REGION Network 10
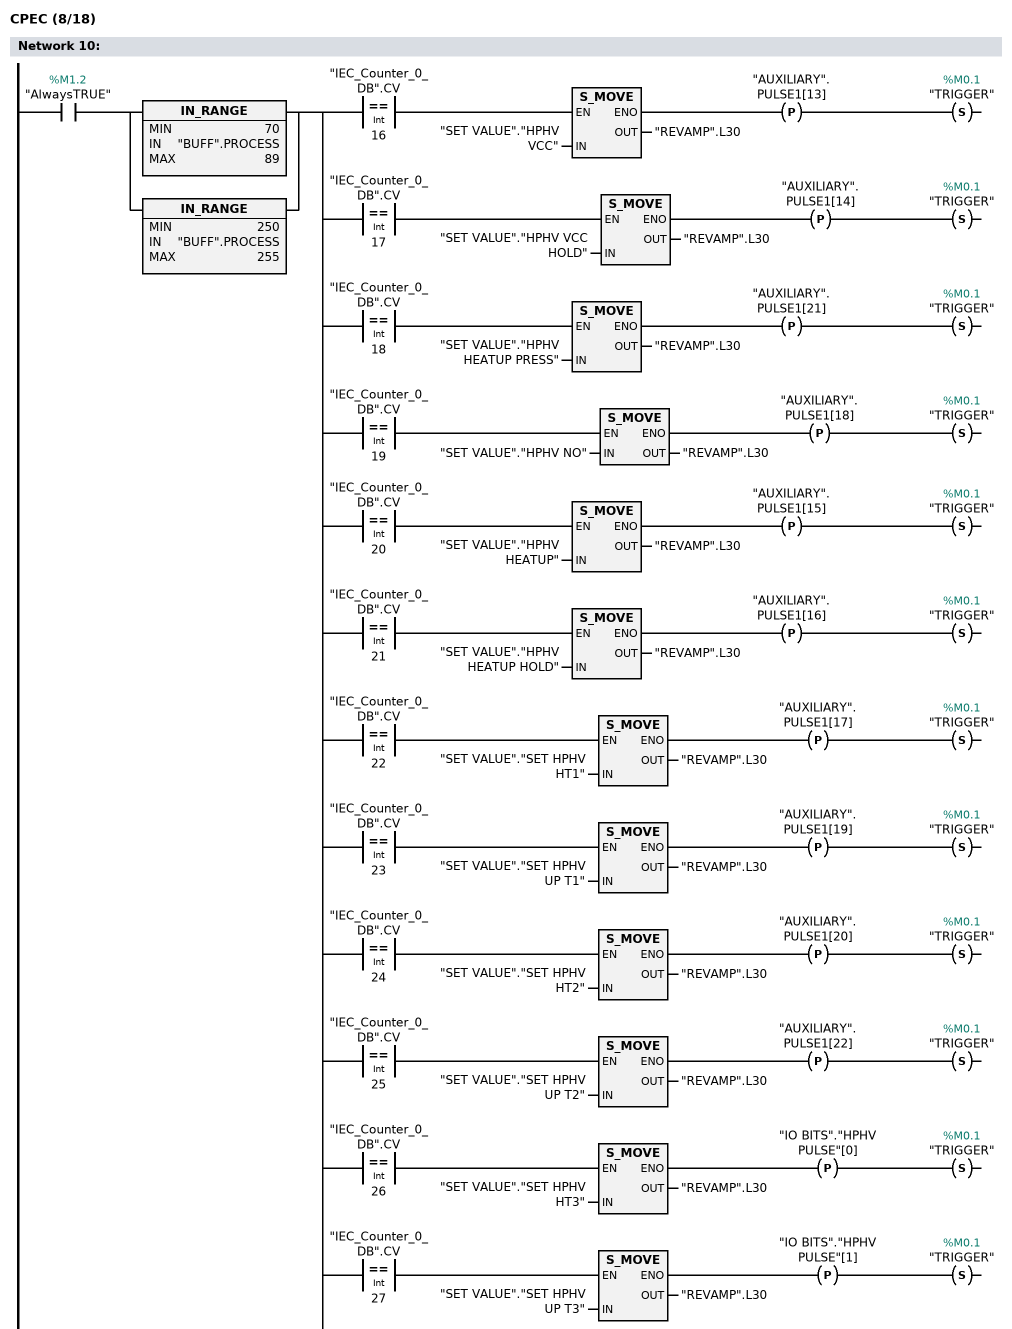
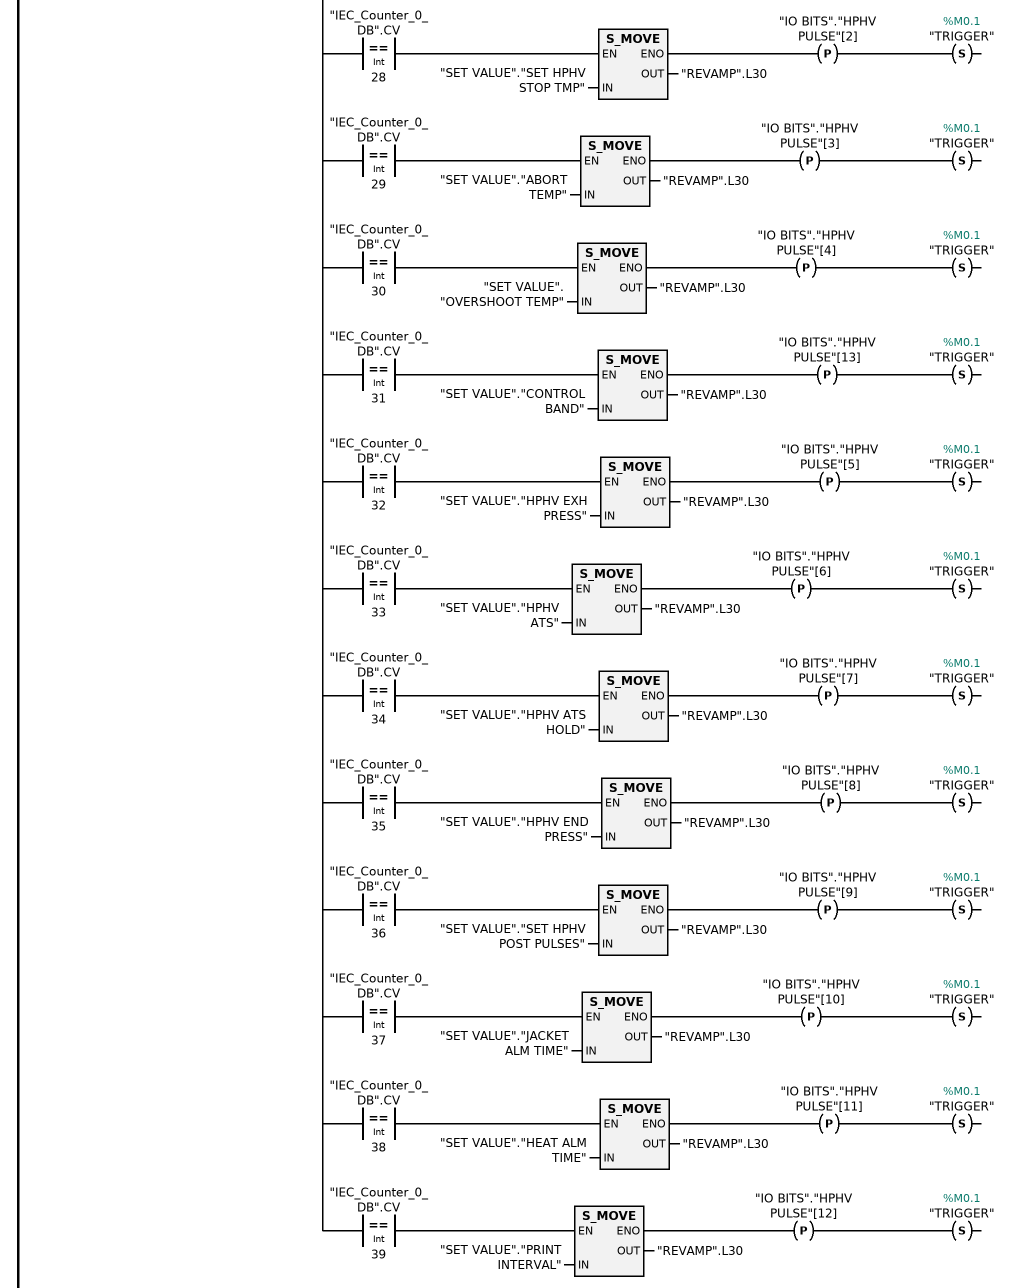
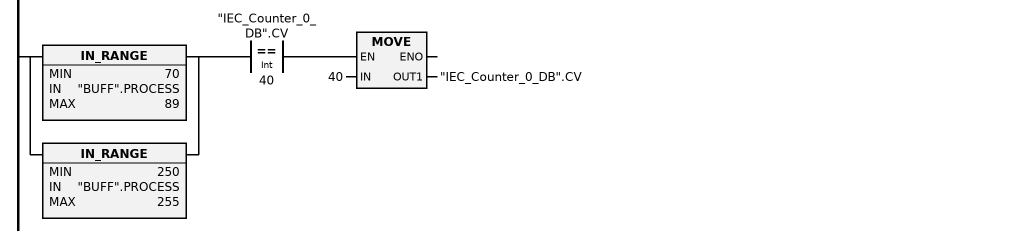
   RUNG wire#powerrail
      Contact( "AlwaysTRUE" )
      wire#w1
      { S7_Templates := "SrcType := Int" } InRange(min := 70, in := "BUFF".PROCESS, max := 89)
      wire#w2
      { S7_Templates := "SrcType := Int" } EQ_Contact(in1 := "IEC_Counter_0_DB".CV, in2 := 16)
      S_Move(in := "SET VALUE"."HPHV VCC", out => "REVAMP".L30)
      P_Trig( "AUXILIARY".PULSE1[13] )
      S_Coil( "TRIGGER" )
   END_RUNG
   RUNG wire#w1
      { S7_Templates := "SrcType := Int" } InRange(min := 250, in := "BUFF".PROCESS, max := 255)
   END_RUNG wire#w2
   RUNG wire#w2
      { S7_Templates := "SrcType := Int" } EQ_Contact(in1 := "IEC_Counter_0_DB".CV, in2 := 17)
      S_Move(in := "SET VALUE"."HPHV VCC HOLD", out => "REVAMP".L30)
      P_Trig( "AUXILIARY".PULSE1[14] )
      S_Coil( "TRIGGER" )
   END_RUNG
   RUNG wire#w2
      { S7_Templates := "SrcType := Int" } EQ_Contact(in1 := "IEC_Counter_0_DB".CV, in2 := 18)
      S_Move(in := "SET VALUE"."HPHV HEATUP PRESS", out => "REVAMP".L30)
      P_Trig( "AUXILIARY".PULSE1[21] )
      S_Coil( "TRIGGER" )
   END_RUNG
   RUNG wire#w2
      { S7_Templates := "SrcType := Int" } EQ_Contact(in1 := "IEC_Counter_0_DB".CV, in2 := 19)
      S_Move(in := "SET VALUE"."HPHV NO", out => "REVAMP".L30)
      P_Trig( "AUXILIARY".PULSE1[18] )
      S_Coil( "TRIGGER" )
   END_RUNG
   RUNG wire#w2
      { S7_Templates := "SrcType := Int" } EQ_Contact(in1 := "IEC_Counter_0_DB".CV, in2 := 20)
      S_Move(in := "SET VALUE"."HPHV HEATUP", out => "REVAMP".L30)
      P_Trig( "AUXILIARY".PULSE1[15] )
      S_Coil( "TRIGGER" )
   END_RUNG
   RUNG wire#w2
      { S7_Templates := "SrcType := Int" } EQ_Contact(in1 := "IEC_Counter_0_DB".CV, in2 := 21)
      S_Move(in := "SET VALUE"."HPHV HEATUP HOLD", out => "REVAMP".L30)
      P_Trig( "AUXILIARY".PULSE1[16] )
      S_Coil( "TRIGGER" )
   END_RUNG
   RUNG wire#w2
      { S7_Templates := "SrcType := Int" } EQ_Contact(in1 := "IEC_Counter_0_DB".CV, in2 := 22)
      S_Move(in := "SET VALUE"."SET HPHV HT1", out => "REVAMP".L30)
      P_Trig( "AUXILIARY".PULSE1[17] )
      S_Coil( "TRIGGER" )
   END_RUNG
   RUNG wire#w2
      { S7_Templates := "SrcType := Int" } EQ_Contact(in1 := "IEC_Counter_0_DB".CV, in2 := 23)
      S_Move(in := "SET VALUE"."SET HPHV UP T1", out => "REVAMP".L30)
      P_Trig( "AUXILIARY".PULSE1[19] )
      S_Coil( "TRIGGER" )
   END_RUNG
   RUNG wire#w2
      { S7_Templates := "SrcType := Int" } EQ_Contact(in1 := "IEC_Counter_0_DB".CV, in2 := 24)
      S_Move(in := "SET VALUE"."SET HPHV HT2", out => "REVAMP".L30)
      P_Trig( "AUXILIARY".PULSE1[20] )
      S_Coil( "TRIGGER" )
   END_RUNG
   RUNG wire#w2
      { S7_Templates := "SrcType := Int" } EQ_Contact(in1 := "IEC_Counter_0_DB".CV, in2 := 25)
      S_Move(in := "SET VALUE"."SET HPHV UP T2", out => "REVAMP".L30)
      P_Trig( "AUXILIARY".PULSE1[22] )
      S_Coil( "TRIGGER" )
   END_RUNG
   RUNG wire#w2
      { S7_Templates := "SrcType := Int" } EQ_Contact(in1 := "IEC_Counter_0_DB".CV, in2 := 26)
      S_Move(in := "SET VALUE"."SET HPHV HT3", out => "REVAMP".L30)
      P_Trig( "IO BITS"."HPHV PULSE"[0] )
      S_Coil( "TRIGGER" )
   END_RUNG
   RUNG wire#w2
      { S7_Templates := "SrcType := Int" } EQ_Contact(in1 := "IEC_Counter_0_DB".CV, in2 := 27)
      S_Move(in := "SET VALUE"."SET HPHV UP T3", out => "REVAMP".L30)
      P_Trig( "IO BITS"."HPHV PULSE"[1] )
      S_Coil( "TRIGGER" )
   END_RUNG
   RUNG wire#w2
      { S7_Templates := "SrcType := Int" } EQ_Contact(in1 := "IEC_Counter_0_DB".CV, in2 := 28)
      S_Move(in := "SET VALUE"."SET HPHV STOP TMP", out => "REVAMP".L30)
      P_Trig( "IO BITS"."HPHV PULSE"[2] )
      S_Coil( "TRIGGER" )
   END_RUNG
   RUNG wire#w2
      { S7_Templates := "SrcType := Int" } EQ_Contact(in1 := "IEC_Counter_0_DB".CV, in2 := 29)
      S_Move(in := "SET VALUE"."ABORT TEMP", out => "REVAMP".L30)
      P_Trig( "IO BITS"."HPHV PULSE"[3] )
      S_Coil( "TRIGGER" )
   END_RUNG
   RUNG wire#w2
      { S7_Templates := "SrcType := Int" } EQ_Contact(in1 := "IEC_Counter_0_DB".CV, in2 := 30)
      S_Move(in := "SET VALUE"."OVERSHOOT TEMP", out => "REVAMP".L30)
      P_Trig( "IO BITS"."HPHV PULSE"[4] )
      S_Coil( "TRIGGER" )
   END_RUNG
   RUNG wire#w2
      { S7_Templates := "SrcType := Int" } EQ_Contact(in1 := "IEC_Counter_0_DB".CV, in2 := 31)
      S_Move(in := "SET VALUE"."CONTROL BAND", out => "REVAMP".L30)
      P_Trig( "IO BITS"."HPHV PULSE"[13] )
      S_Coil( "TRIGGER" )
   END_RUNG
   RUNG wire#w2
      { S7_Templates := "SrcType := Int" } EQ_Contact(in1 := "IEC_Counter_0_DB".CV, in2 := 32)
      S_Move(in := "SET VALUE"."HPHV EXH PRESS", out => "REVAMP".L30)
      P_Trig( "IO BITS"."HPHV PULSE"[5] )
      S_Coil( "TRIGGER" )
   END_RUNG
   RUNG wire#w2
      { S7_Templates := "SrcType := Int" } EQ_Contact(in1 := "IEC_Counter_0_DB".CV, in2 := 33)
      S_Move(in := "SET VALUE"."HPHV ATS", out => "REVAMP".L30)
      P_Trig( "IO BITS"."HPHV PULSE"[6] )
      S_Coil( "TRIGGER" )
   END_RUNG
   RUNG wire#w2
      { S7_Templates := "SrcType := Int" } EQ_Contact(in1 := "IEC_Counter_0_DB".CV, in2 := 34)
      S_Move(in := "SET VALUE"."HPHV ATS HOLD", out => "REVAMP".L30)
      P_Trig( "IO BITS"."HPHV PULSE"[7] )
      S_Coil( "TRIGGER" )
   END_RUNG
   RUNG wire#w2
      { S7_Templates := "SrcType := Int" } EQ_Contact(in1 := "IEC_Counter_0_DB".CV, in2 := 35)
      S_Move(in := "SET VALUE"."HPHV END PRESS", out => "REVAMP".L30)
      P_Trig( "IO BITS"."HPHV PULSE"[8] )
      S_Coil( "TRIGGER" )
   END_RUNG
   RUNG wire#w2
      { S7_Templates := "SrcType := Int" } EQ_Contact(in1 := "IEC_Counter_0_DB".CV, in2 := 36)
      S_Move(in := "SET VALUE"."SET HPHV POST PULSES", out => "REVAMP".L30)
      P_Trig( "IO BITS"."HPHV PULSE"[9] )
      S_Coil( "TRIGGER" )
   END_RUNG
   RUNG wire#w2
      { S7_Templates := "SrcType := Int" } EQ_Contact(in1 := "IEC_Counter_0_DB".CV, in2 := 37)
      S_Move(in := "SET VALUE"."JACKET ALM TIME", out => "REVAMP".L30)
      P_Trig( "IO BITS"."HPHV PULSE"[10] )
      S_Coil( "TRIGGER" )
   END_RUNG
   RUNG wire#w2
      { S7_Templates := "SrcType := Int" } EQ_Contact(in1 := "IEC_Counter_0_DB".CV, in2 := 38)
      S_Move(in := "SET VALUE"."HEAT ALM TIME", out => "REVAMP".L30)
      P_Trig( "IO BITS"."HPHV PULSE"[11] )
      S_Coil( "TRIGGER" )
   END_RUNG
   RUNG wire#w2
      { S7_Templates := "SrcType := Int" } EQ_Contact(in1 := "IEC_Counter_0_DB".CV, in2 := 39)
      S_Move(in := "SET VALUE"."PRINT INTERVAL", out => "REVAMP".L30)
      P_Trig( "IO BITS"."HPHV PULSE"[12] )
      S_Coil( "TRIGGER" )
   END_RUNG
   RUNG wire#powerrail
      { S7_Templates := "SrcType := Int" } InRange(min := 70, in := "BUFF".PROCESS, max := 89)
      wire#w3
      { S7_Templates := "SrcType := Int" } EQ_Contact(in1 := "IEC_Counter_0_DB".CV, in2 := 40)
      Move(in := 40, out1 => "IEC_Counter_0_DB".CV)
   END_RUNG
   RUNG wire#powerrail
      { S7_Templates := "SrcType := Int" } InRange(min := 250, in := "BUFF".PROCESS, max := 255)
   END_RUNG wire#w3
   // the same network as SCL:
   #_w1 := "AlwaysTRUE" AND (((70 <= "BUFF".PROCESS) AND ("BUFF".PROCESS <= 89)) OR ((250 <= "BUFF".PROCESS) AND ("BUFF".PROCESS <= 255)));
   #_w2 := #_w1 AND ("IEC_Counter_0_DB".CV = 16);
   IF #_w2 THEN "REVAMP".L30 := "SET VALUE"."HPHV VCC"; END_IF;
   #_w3 := #_w2 AND NOT "AUXILIARY".PULSE1[13];   // rising edge
   "AUXILIARY".PULSE1[13] := #_w2;
   IF #_w3 THEN "TRIGGER" := TRUE; END_IF;
   #_w4 := #_w1 AND ("IEC_Counter_0_DB".CV = 17);
   IF #_w4 THEN "REVAMP".L30 := "SET VALUE"."HPHV VCC HOLD"; END_IF;
   #_w5 := #_w4 AND NOT "AUXILIARY".PULSE1[14];   // rising edge
   "AUXILIARY".PULSE1[14] := #_w4;
   IF #_w5 THEN "TRIGGER" := TRUE; END_IF;
   #_w6 := #_w1 AND ("IEC_Counter_0_DB".CV = 18);
   IF #_w6 THEN "REVAMP".L30 := "SET VALUE"."HPHV HEATUP PRESS"; END_IF;
   #_w7 := #_w6 AND NOT "AUXILIARY".PULSE1[21];   // rising edge
   "AUXILIARY".PULSE1[21] := #_w6;
   IF #_w7 THEN "TRIGGER" := TRUE; END_IF;
   #_w8 := #_w1 AND ("IEC_Counter_0_DB".CV = 19);
   IF #_w8 THEN "REVAMP".L30 := "SET VALUE"."HPHV NO"; END_IF;
   #_w9 := #_w8 AND NOT "AUXILIARY".PULSE1[18];   // rising edge
   "AUXILIARY".PULSE1[18] := #_w8;
   IF #_w9 THEN "TRIGGER" := TRUE; END_IF;
   #_w10 := #_w1 AND ("IEC_Counter_0_DB".CV = 20);
   IF #_w10 THEN "REVAMP".L30 := "SET VALUE"."HPHV HEATUP"; END_IF;
   #_w11 := #_w10 AND NOT "AUXILIARY".PULSE1[15];   // rising edge
   "AUXILIARY".PULSE1[15] := #_w10;
   IF #_w11 THEN "TRIGGER" := TRUE; END_IF;
   #_w12 := #_w1 AND ("IEC_Counter_0_DB".CV = 21);
   IF #_w12 THEN "REVAMP".L30 := "SET VALUE"."HPHV HEATUP HOLD"; END_IF;
   #_w13 := #_w12 AND NOT "AUXILIARY".PULSE1[16];   // rising edge
   "AUXILIARY".PULSE1[16] := #_w12;
   IF #_w13 THEN "TRIGGER" := TRUE; END_IF;
   #_w14 := #_w1 AND ("IEC_Counter_0_DB".CV = 22);
   IF #_w14 THEN "REVAMP".L30 := "SET VALUE"."SET HPHV HT1"; END_IF;
   #_w15 := #_w14 AND NOT "AUXILIARY".PULSE1[17];   // rising edge
   "AUXILIARY".PULSE1[17] := #_w14;
   IF #_w15 THEN "TRIGGER" := TRUE; END_IF;
   #_w16 := #_w1 AND ("IEC_Counter_0_DB".CV = 23);
   IF #_w16 THEN "REVAMP".L30 := "SET VALUE"."SET HPHV UP T1"; END_IF;
   #_w17 := #_w16 AND NOT "AUXILIARY".PULSE1[19];   // rising edge
   "AUXILIARY".PULSE1[19] := #_w16;
   IF #_w17 THEN "TRIGGER" := TRUE; END_IF;
   #_w18 := #_w1 AND ("IEC_Counter_0_DB".CV = 24);
   IF #_w18 THEN "REVAMP".L30 := "SET VALUE"."SET HPHV HT2"; END_IF;
   #_w19 := #_w18 AND NOT "AUXILIARY".PULSE1[20];   // rising edge
   "AUXILIARY".PULSE1[20] := #_w18;
   IF #_w19 THEN "TRIGGER" := TRUE; END_IF;
   #_w20 := #_w1 AND ("IEC_Counter_0_DB".CV = 25);
   IF #_w20 THEN "REVAMP".L30 := "SET VALUE"."SET HPHV UP T2"; END_IF;
   #_w21 := #_w20 AND NOT "AUXILIARY".PULSE1[22];   // rising edge
   "AUXILIARY".PULSE1[22] := #_w20;
   IF #_w21 THEN "TRIGGER" := TRUE; END_IF;
   #_w22 := #_w1 AND ("IEC_Counter_0_DB".CV = 26);
   IF #_w22 THEN "REVAMP".L30 := "SET VALUE"."SET HPHV HT3"; END_IF;
   #_w23 := #_w22 AND NOT "IO BITS"."HPHV PULSE"[0];   // rising edge
   "IO BITS"."HPHV PULSE"[0] := #_w22;
   IF #_w23 THEN "TRIGGER" := TRUE; END_IF;
   #_w24 := #_w1 AND ("IEC_Counter_0_DB".CV = 27);
   IF #_w24 THEN "REVAMP".L30 := "SET VALUE"."SET HPHV UP T3"; END_IF;
   #_w25 := #_w24 AND NOT "IO BITS"."HPHV PULSE"[1];   // rising edge
   "IO BITS"."HPHV PULSE"[1] := #_w24;
   IF #_w25 THEN "TRIGGER" := TRUE; END_IF;
   #_w26 := #_w1 AND ("IEC_Counter_0_DB".CV = 28);
   IF #_w26 THEN "REVAMP".L30 := "SET VALUE"."SET HPHV STOP TMP"; END_IF;
   #_w27 := #_w26 AND NOT "IO BITS"."HPHV PULSE"[2];   // rising edge
   "IO BITS"."HPHV PULSE"[2] := #_w26;
   IF #_w27 THEN "TRIGGER" := TRUE; END_IF;
   #_w28 := #_w1 AND ("IEC_Counter_0_DB".CV = 29);
   IF #_w28 THEN "REVAMP".L30 := "SET VALUE"."ABORT TEMP"; END_IF;
   #_w29 := #_w28 AND NOT "IO BITS"."HPHV PULSE"[3];   // rising edge
   "IO BITS"."HPHV PULSE"[3] := #_w28;
   IF #_w29 THEN "TRIGGER" := TRUE; END_IF;
   #_w30 := #_w1 AND ("IEC_Counter_0_DB".CV = 30);
   IF #_w30 THEN "REVAMP".L30 := "SET VALUE"."OVERSHOOT TEMP"; END_IF;
   #_w31 := #_w30 AND NOT "IO BITS"."HPHV PULSE"[4];   // rising edge
   "IO BITS"."HPHV PULSE"[4] := #_w30;
   IF #_w31 THEN "TRIGGER" := TRUE; END_IF;
   #_w32 := #_w1 AND ("IEC_Counter_0_DB".CV = 31);
   IF #_w32 THEN "REVAMP".L30 := "SET VALUE"."CONTROL BAND"; END_IF;
   #_w33 := #_w32 AND NOT "IO BITS"."HPHV PULSE"[13];   // rising edge
   "IO BITS"."HPHV PULSE"[13] := #_w32;
   IF #_w33 THEN "TRIGGER" := TRUE; END_IF;
   #_w34 := #_w1 AND ("IEC_Counter_0_DB".CV = 32);
   IF #_w34 THEN "REVAMP".L30 := "SET VALUE"."HPHV EXH PRESS"; END_IF;
   #_w35 := #_w34 AND NOT "IO BITS"."HPHV PULSE"[5];   // rising edge
   "IO BITS"."HPHV PULSE"[5] := #_w34;
   IF #_w35 THEN "TRIGGER" := TRUE; END_IF;
   #_w36 := #_w1 AND ("IEC_Counter_0_DB".CV = 33);
   IF #_w36 THEN "REVAMP".L30 := "SET VALUE"."HPHV ATS"; END_IF;
   #_w37 := #_w36 AND NOT "IO BITS"."HPHV PULSE"[6];   // rising edge
   "IO BITS"."HPHV PULSE"[6] := #_w36;
   IF #_w37 THEN "TRIGGER" := TRUE; END_IF;
   #_w38 := #_w1 AND ("IEC_Counter_0_DB".CV = 34);
   IF #_w38 THEN "REVAMP".L30 := "SET VALUE"."HPHV ATS HOLD"; END_IF;
   #_w39 := #_w38 AND NOT "IO BITS"."HPHV PULSE"[7];   // rising edge
   "IO BITS"."HPHV PULSE"[7] := #_w38;
   IF #_w39 THEN "TRIGGER" := TRUE; END_IF;
   #_w40 := #_w1 AND ("IEC_Counter_0_DB".CV = 35);
   IF #_w40 THEN "REVAMP".L30 := "SET VALUE"."HPHV END PRESS"; END_IF;
   #_w41 := #_w40 AND NOT "IO BITS"."HPHV PULSE"[8];   // rising edge
   "IO BITS"."HPHV PULSE"[8] := #_w40;
   IF #_w41 THEN "TRIGGER" := TRUE; END_IF;
   #_w42 := #_w1 AND ("IEC_Counter_0_DB".CV = 36);
   IF #_w42 THEN "REVAMP".L30 := "SET VALUE"."SET HPHV POST PULSES"; END_IF;
   #_w43 := #_w42 AND NOT "IO BITS"."HPHV PULSE"[9];   // rising edge
   "IO BITS"."HPHV PULSE"[9] := #_w42;
   IF #_w43 THEN "TRIGGER" := TRUE; END_IF;
   #_w44 := #_w1 AND ("IEC_Counter_0_DB".CV = 37);
   IF #_w44 THEN "REVAMP".L30 := "SET VALUE"."JACKET ALM TIME"; END_IF;
   #_w45 := #_w44 AND NOT "IO BITS"."HPHV PULSE"[10];   // rising edge
   "IO BITS"."HPHV PULSE"[10] := #_w44;
   IF #_w45 THEN "TRIGGER" := TRUE; END_IF;
   #_w46 := #_w1 AND ("IEC_Counter_0_DB".CV = 38);
   IF #_w46 THEN "REVAMP".L30 := "SET VALUE"."HEAT ALM TIME"; END_IF;
   #_w47 := #_w46 AND NOT "IO BITS"."HPHV PULSE"[11];   // rising edge
   "IO BITS"."HPHV PULSE"[11] := #_w46;
   IF #_w47 THEN "TRIGGER" := TRUE; END_IF;
   #_w48 := #_w1 AND ("IEC_Counter_0_DB".CV = 39);
   IF #_w48 THEN "REVAMP".L30 := "SET VALUE"."PRINT INTERVAL"; END_IF;
   #_w49 := #_w48 AND NOT "IO BITS"."HPHV PULSE"[12];   // rising edge
   "IO BITS"."HPHV PULSE"[12] := #_w48;
   IF #_w49 THEN "TRIGGER" := TRUE; END_IF;
   IF (((70 <= "BUFF".PROCESS) AND ("BUFF".PROCESS <= 89)) OR ((250 <= "BUFF".PROCESS) AND ("BUFF".PROCESS <= 255))) AND ("IEC_Counter_0_DB".CV = 40) THEN
       "IEC_Counter_0_DB".CV := 40;
   END_IF;
END_REGION

REGION Network 11
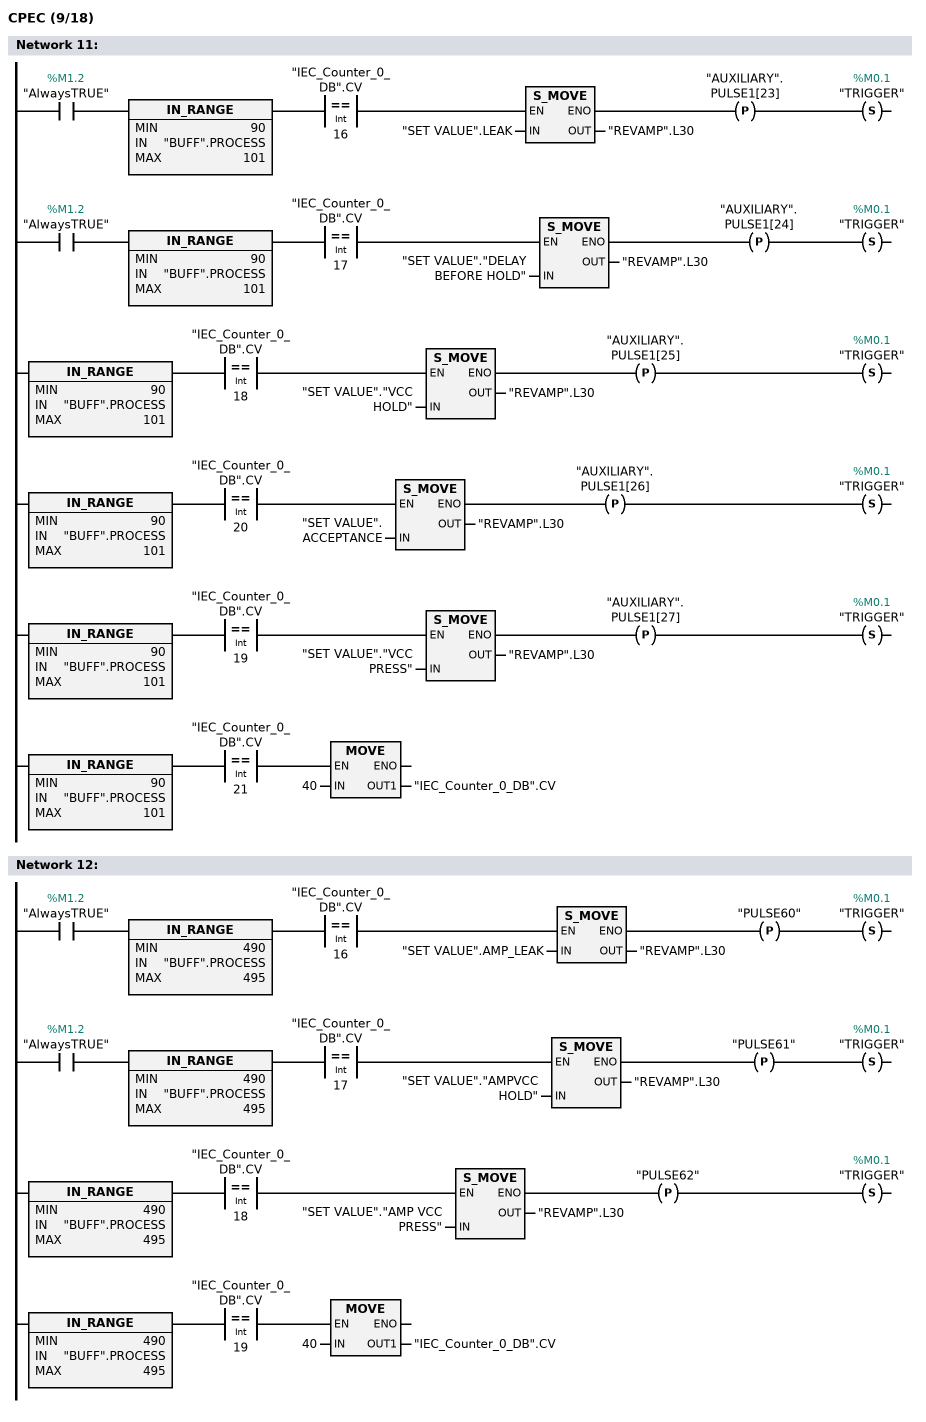
   RUNG wire#powerrail
      Contact( "AlwaysTRUE" )
      { S7_Templates := "SrcType := Int" } InRange(min := 90, in := "BUFF".PROCESS, max := 101)
      { S7_Templates := "SrcType := Int" } EQ_Contact(in1 := "IEC_Counter_0_DB".CV, in2 := 16)
      S_Move(in := "SET VALUE".LEAK, out => "REVAMP".L30)
      P_Trig( "AUXILIARY".PULSE1[23] )
      S_Coil( "TRIGGER" )
   END_RUNG
   RUNG wire#powerrail
      Contact( "AlwaysTRUE" )
      { S7_Templates := "SrcType := Int" } InRange(min := 90, in := "BUFF".PROCESS, max := 101)
      { S7_Templates := "SrcType := Int" } EQ_Contact(in1 := "IEC_Counter_0_DB".CV, in2 := 17)
      S_Move(in := "SET VALUE"."DELAY BEFORE HOLD", out => "REVAMP".L30)
      P_Trig( "AUXILIARY".PULSE1[24] )
      S_Coil( "TRIGGER" )
   END_RUNG
   RUNG wire#powerrail
      { S7_Templates := "SrcType := Int" } InRange(min := 90, in := "BUFF".PROCESS, max := 101)
      { S7_Templates := "SrcType := Int" } EQ_Contact(in1 := "IEC_Counter_0_DB".CV, in2 := 18)
      S_Move(in := "SET VALUE"."VCC HOLD", out => "REVAMP".L30)
      P_Trig( "AUXILIARY".PULSE1[25] )
      S_Coil( "TRIGGER" )
   END_RUNG
   RUNG wire#powerrail
      { S7_Templates := "SrcType := Int" } InRange(min := 90, in := "BUFF".PROCESS, max := 101)
      { S7_Templates := "SrcType := Int" } EQ_Contact(in1 := "IEC_Counter_0_DB".CV, in2 := 20)
      S_Move(in := "SET VALUE".ACCEPTANCE, out => "REVAMP".L30)
      P_Trig( "AUXILIARY".PULSE1[26] )
      S_Coil( "TRIGGER" )
   END_RUNG
   RUNG wire#powerrail
      { S7_Templates := "SrcType := Int" } InRange(min := 90, in := "BUFF".PROCESS, max := 101)
      { S7_Templates := "SrcType := Int" } EQ_Contact(in1 := "IEC_Counter_0_DB".CV, in2 := 19)
      S_Move(in := "SET VALUE"."VCC PRESS", out => "REVAMP".L30)
      P_Trig( "AUXILIARY".PULSE1[27] )
      S_Coil( "TRIGGER" )
   END_RUNG
   RUNG wire#powerrail
      { S7_Templates := "SrcType := Int" } InRange(min := 90, in := "BUFF".PROCESS, max := 101)
      { S7_Templates := "SrcType := Int" } EQ_Contact(in1 := "IEC_Counter_0_DB".CV, in2 := 21)
      Move(in := 40, out1 => "IEC_Counter_0_DB".CV)
   END_RUNG
   // the same network as SCL:
   #_w1 := "AlwaysTRUE" AND (90 <= "BUFF".PROCESS) AND ("BUFF".PROCESS <= 101) AND ("IEC_Counter_0_DB".CV = 16);
   IF #_w1 THEN "REVAMP".L30 := "SET VALUE".LEAK; END_IF;
   #_w2 := #_w1 AND NOT "AUXILIARY".PULSE1[23];   // rising edge
   "AUXILIARY".PULSE1[23] := #_w1;
   IF #_w2 THEN "TRIGGER" := TRUE; END_IF;
   #_w3 := "AlwaysTRUE" AND (90 <= "BUFF".PROCESS) AND ("BUFF".PROCESS <= 101) AND ("IEC_Counter_0_DB".CV = 17);
   IF #_w3 THEN "REVAMP".L30 := "SET VALUE"."DELAY BEFORE HOLD"; END_IF;
   #_w4 := #_w3 AND NOT "AUXILIARY".PULSE1[24];   // rising edge
   "AUXILIARY".PULSE1[24] := #_w3;
   IF #_w4 THEN "TRIGGER" := TRUE; END_IF;
   #_w5 := (90 <= "BUFF".PROCESS) AND ("BUFF".PROCESS <= 101) AND ("IEC_Counter_0_DB".CV = 18);
   IF #_w5 THEN "REVAMP".L30 := "SET VALUE"."VCC HOLD"; END_IF;
   #_w6 := #_w5 AND NOT "AUXILIARY".PULSE1[25];   // rising edge
   "AUXILIARY".PULSE1[25] := #_w5;
   IF #_w6 THEN "TRIGGER" := TRUE; END_IF;
   #_w7 := (90 <= "BUFF".PROCESS) AND ("BUFF".PROCESS <= 101) AND ("IEC_Counter_0_DB".CV = 20);
   IF #_w7 THEN "REVAMP".L30 := "SET VALUE".ACCEPTANCE; END_IF;
   #_w8 := #_w7 AND NOT "AUXILIARY".PULSE1[26];   // rising edge
   "AUXILIARY".PULSE1[26] := #_w7;
   IF #_w8 THEN "TRIGGER" := TRUE; END_IF;
   #_w9 := (90 <= "BUFF".PROCESS) AND ("BUFF".PROCESS <= 101) AND ("IEC_Counter_0_DB".CV = 19);
   IF #_w9 THEN "REVAMP".L30 := "SET VALUE"."VCC PRESS"; END_IF;
   #_w10 := #_w9 AND NOT "AUXILIARY".PULSE1[27];   // rising edge
   "AUXILIARY".PULSE1[27] := #_w9;
   IF #_w10 THEN "TRIGGER" := TRUE; END_IF;
   IF (90 <= "BUFF".PROCESS) AND ("BUFF".PROCESS <= 101) AND ("IEC_Counter_0_DB".CV = 21) THEN
       "IEC_Counter_0_DB".CV := 40;
   END_IF;
END_REGION

REGION Network 12
   RUNG wire#powerrail
      Contact( "AlwaysTRUE" )
      { S7_Templates := "SrcType := Int" } InRange(min := 490, in := "BUFF".PROCESS, max := 495)
      { S7_Templates := "SrcType := Int" } EQ_Contact(in1 := "IEC_Counter_0_DB".CV, in2 := 16)
      S_Move(in := "SET VALUE".AMP_LEAK, out => "REVAMP".L30)
      P_Trig( "PULSE60" )
      S_Coil( "TRIGGER" )
   END_RUNG
   RUNG wire#powerrail
      Contact( "AlwaysTRUE" )
      { S7_Templates := "SrcType := Int" } InRange(min := 490, in := "BUFF".PROCESS, max := 495)
      { S7_Templates := "SrcType := Int" } EQ_Contact(in1 := "IEC_Counter_0_DB".CV, in2 := 17)
      S_Move(in := "SET VALUE"."AMPVCC HOLD", out => "REVAMP".L30)
      P_Trig( "PULSE61" )
      S_Coil( "TRIGGER" )
   END_RUNG
   RUNG wire#powerrail
      { S7_Templates := "SrcType := Int" } InRange(min := 490, in := "BUFF".PROCESS, max := 495)
      { S7_Templates := "SrcType := Int" } EQ_Contact(in1 := "IEC_Counter_0_DB".CV, in2 := 18)
      S_Move(in := "SET VALUE"."AMP VCC PRESS", out => "REVAMP".L30)
      P_Trig( "PULSE62" )
      S_Coil( "TRIGGER" )
   END_RUNG
   RUNG wire#powerrail
      { S7_Templates := "SrcType := Int" } InRange(min := 490, in := "BUFF".PROCESS, max := 495)
      { S7_Templates := "SrcType := Int" } EQ_Contact(in1 := "IEC_Counter_0_DB".CV, in2 := 19)
      Move(in := 40, out1 => "IEC_Counter_0_DB".CV)
   END_RUNG
   // the same network as SCL:
   #_w1 := "AlwaysTRUE" AND (490 <= "BUFF".PROCESS) AND ("BUFF".PROCESS <= 495) AND ("IEC_Counter_0_DB".CV = 16);
   IF #_w1 THEN "REVAMP".L30 := "SET VALUE".AMP_LEAK; END_IF;
   #_w2 := #_w1 AND NOT "PULSE60";   // rising edge
   "PULSE60" := #_w1;
   IF #_w2 THEN "TRIGGER" := TRUE; END_IF;
   #_w3 := "AlwaysTRUE" AND (490 <= "BUFF".PROCESS) AND ("BUFF".PROCESS <= 495) AND ("IEC_Counter_0_DB".CV = 17);
   IF #_w3 THEN "REVAMP".L30 := "SET VALUE"."AMPVCC HOLD"; END_IF;
   #_w4 := #_w3 AND NOT "PULSE61";   // rising edge
   "PULSE61" := #_w3;
   IF #_w4 THEN "TRIGGER" := TRUE; END_IF;
   #_w5 := (490 <= "BUFF".PROCESS) AND ("BUFF".PROCESS <= 495) AND ("IEC_Counter_0_DB".CV = 18);
   IF #_w5 THEN "REVAMP".L30 := "SET VALUE"."AMP VCC PRESS"; END_IF;
   #_w6 := #_w5 AND NOT "PULSE62";   // rising edge
   "PULSE62" := #_w5;
   IF #_w6 THEN "TRIGGER" := TRUE; END_IF;
   IF (490 <= "BUFF".PROCESS) AND ("BUFF".PROCESS <= 495) AND ("IEC_Counter_0_DB".CV = 19) THEN
       "IEC_Counter_0_DB".CV := 40;
   END_IF;
END_REGION

REGION Network 13
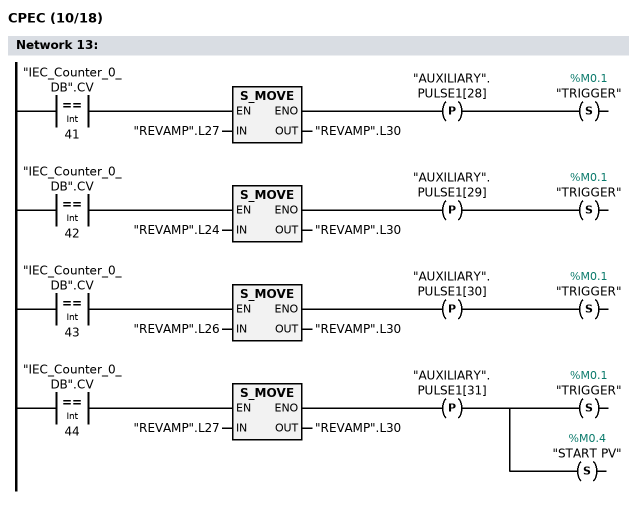
   RUNG wire#powerrail
      { S7_Templates := "SrcType := Int" } EQ_Contact(in1 := "IEC_Counter_0_DB".CV, in2 := 41)
      S_Move(in := "REVAMP".L27, out => "REVAMP".L30)
      P_Trig( "AUXILIARY".PULSE1[28] )
      S_Coil( "TRIGGER" )
   END_RUNG
   RUNG wire#powerrail
      { S7_Templates := "SrcType := Int" } EQ_Contact(in1 := "IEC_Counter_0_DB".CV, in2 := 42)
      S_Move(in := "REVAMP".L24, out => "REVAMP".L30)
      P_Trig( "AUXILIARY".PULSE1[29] )
      S_Coil( "TRIGGER" )
   END_RUNG
   RUNG wire#powerrail
      { S7_Templates := "SrcType := Int" } EQ_Contact(in1 := "IEC_Counter_0_DB".CV, in2 := 43)
      S_Move(in := "REVAMP".L26, out => "REVAMP".L30)
      P_Trig( "AUXILIARY".PULSE1[30] )
      S_Coil( "TRIGGER" )
   END_RUNG
   RUNG wire#powerrail
      { S7_Templates := "SrcType := Int" } EQ_Contact(in1 := "IEC_Counter_0_DB".CV, in2 := 44)
      S_Move(in := "REVAMP".L27, out => "REVAMP".L30)
      P_Trig( "AUXILIARY".PULSE1[31] )
      wire#w1
      S_Coil( "TRIGGER" )
   END_RUNG
   RUNG wire#w1
      S_Coil( "START PV" )
   END_RUNG
   // the same network as SCL:
   #_w1 := "IEC_Counter_0_DB".CV = 41;
   IF #_w1 THEN "REVAMP".L30 := "REVAMP".L27; END_IF;
   #_w2 := #_w1 AND NOT "AUXILIARY".PULSE1[28];   // rising edge
   "AUXILIARY".PULSE1[28] := #_w1;
   IF #_w2 THEN "TRIGGER" := TRUE; END_IF;
   #_w3 := "IEC_Counter_0_DB".CV = 42;
   IF #_w3 THEN "REVAMP".L30 := "REVAMP".L24; END_IF;
   #_w4 := #_w3 AND NOT "AUXILIARY".PULSE1[29];   // rising edge
   "AUXILIARY".PULSE1[29] := #_w3;
   IF #_w4 THEN "TRIGGER" := TRUE; END_IF;
   #_w5 := "IEC_Counter_0_DB".CV = 43;
   IF #_w5 THEN "REVAMP".L30 := "REVAMP".L26; END_IF;
   #_w6 := #_w5 AND NOT "AUXILIARY".PULSE1[30];   // rising edge
   "AUXILIARY".PULSE1[30] := #_w5;
   IF #_w6 THEN "TRIGGER" := TRUE; END_IF;
   #_w7 := "IEC_Counter_0_DB".CV = 44;
   IF #_w7 THEN "REVAMP".L30 := "REVAMP".L27; END_IF;
   #_w8 := #_w7 AND NOT "AUXILIARY".PULSE1[31];   // rising edge
   "AUXILIARY".PULSE1[31] := #_w7;
   IF #_w8 THEN
       "TRIGGER" := TRUE;
       "START PV" := TRUE;
   END_IF;
END_REGION

REGION Network 15
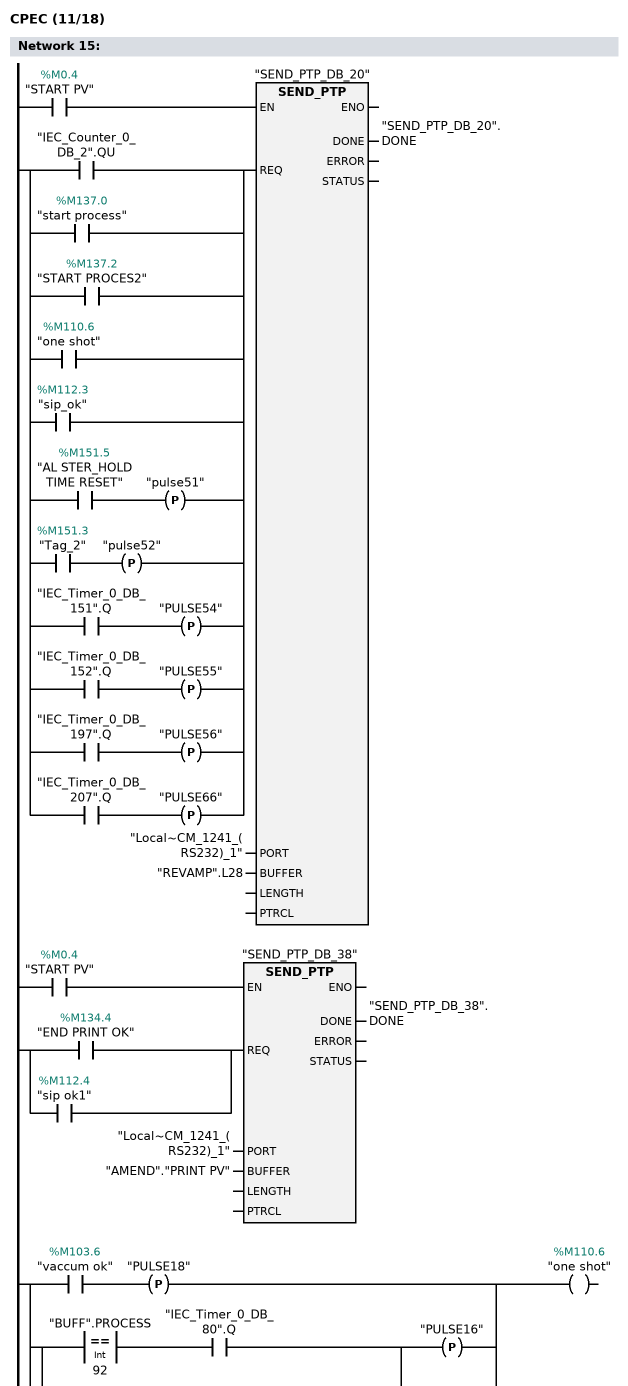
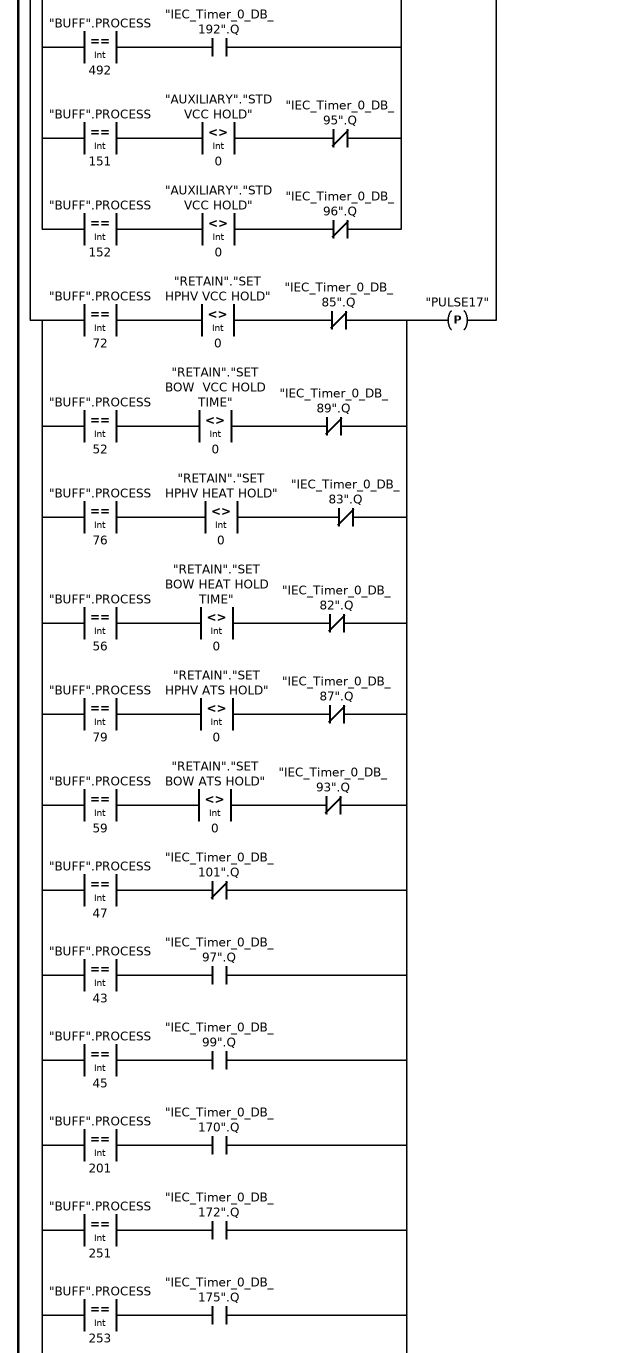
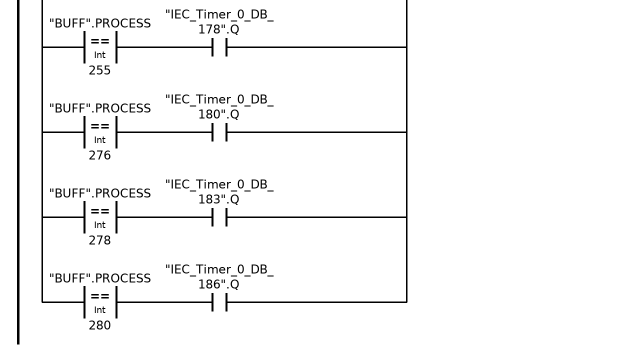
   RUNG wire#powerrail
      Contact( "START PV" )
      "SEND_PTP_DB_20".SEND_PTP(REQ := wire#w1, PORT := "Local~CM_1241_(RS232)_1", BUFFER := "REVAMP".L28, LENGTH :=, PTRCL :=, DONE => "SEND_PTP_DB_20".DONE, ERROR =>, STATUS =>)
   END_RUNG
   RUNG wire#powerrail
      Contact( "IEC_Counter_0_DB_2".QU )
   END_RUNG wire#w1
   RUNG wire#powerrail
      Contact( "start process" )
   END_RUNG wire#w1
   RUNG wire#powerrail
      Contact( "START PROCES2" )
   END_RUNG wire#w1
   RUNG wire#powerrail
      Contact( "one shot" )
   END_RUNG wire#w1
   RUNG wire#powerrail
      Contact( "sip_ok" )
   END_RUNG wire#w1
   RUNG wire#powerrail
      Contact( "AL STER_HOLD TIME RESET" )
      P_Trig( "pulse51" )
   END_RUNG wire#w1
   RUNG wire#powerrail
      Contact( "Tag_2" )
      P_Trig( "pulse52" )
   END_RUNG wire#w1
   RUNG wire#powerrail
      Contact( "IEC_Timer_0_DB_151".Q )
      P_Trig( "PULSE54" )
   END_RUNG wire#w1
   RUNG wire#powerrail
      Contact( "IEC_Timer_0_DB_152".Q )
      P_Trig( "PULSE55" )
   END_RUNG wire#w1
   RUNG wire#powerrail
      Contact( "IEC_Timer_0_DB_197".Q )
      P_Trig( "PULSE56" )
   END_RUNG wire#w1
   RUNG wire#powerrail
      Contact( "IEC_Timer_0_DB_207".Q )
      P_Trig( "PULSE66" )
   END_RUNG wire#w1
   RUNG wire#powerrail
      Contact( "START PV" )
      "SEND_PTP_DB_38".SEND_PTP(REQ := wire#w2, PORT := "Local~CM_1241_(RS232)_1", BUFFER := "AMEND"."PRINT PV", LENGTH :=, PTRCL :=, DONE => "SEND_PTP_DB_38".DONE, ERROR =>, STATUS =>)
   END_RUNG
   RUNG wire#powerrail
      Contact( "END PRINT OK" )
   END_RUNG wire#w2
   RUNG wire#powerrail
      Contact( "sip ok1" )
   END_RUNG wire#w2
   RUNG wire#powerrail
      Contact( "vaccum ok" )
      P_Trig( "PULSE18" )
      wire#w3
      Coil( "one shot" )
   END_RUNG
   RUNG wire#powerrail
      { S7_Templates := "SrcType := Int" } EQ_Contact(in1 := "BUFF".PROCESS, in2 := 92)
      Contact( "IEC_Timer_0_DB_80".Q )
      wire#w4
      P_Trig( "PULSE16" )
   END_RUNG wire#w3
   RUNG wire#powerrail
      { S7_Templates := "SrcType := Int" } EQ_Contact(in1 := "BUFF".PROCESS, in2 := 492)
      Contact( "IEC_Timer_0_DB_192".Q )
   END_RUNG wire#w4
   RUNG wire#powerrail
      { S7_Templates := "SrcType := Int" } EQ_Contact(in1 := "BUFF".PROCESS, in2 := 151)
      { S7_Templates := "SrcType := Int" } NE_Contact(in1 := "AUXILIARY"."STD VCC HOLD", in2 := 0)
      I_Contact( "IEC_Timer_0_DB_95".Q )
   END_RUNG wire#w4
   RUNG wire#powerrail
      { S7_Templates := "SrcType := Int" } EQ_Contact(in1 := "BUFF".PROCESS, in2 := 152)
      { S7_Templates := "SrcType := Int" } NE_Contact(in1 := "AUXILIARY"."STD VCC HOLD", in2 := 0)
      I_Contact( "IEC_Timer_0_DB_96".Q )
   END_RUNG wire#w4
   RUNG wire#powerrail
      { S7_Templates := "SrcType := Int" } EQ_Contact(in1 := "BUFF".PROCESS, in2 := 72)
      { S7_Templates := "SrcType := Int" } NE_Contact(in1 := "RETAIN"."SET HPHV VCC HOLD", in2 := 0)
      I_Contact( "IEC_Timer_0_DB_85".Q )
      wire#w5
      P_Trig( "PULSE17" )
   END_RUNG wire#w3
   RUNG wire#powerrail
      { S7_Templates := "SrcType := Int" } EQ_Contact(in1 := "BUFF".PROCESS, in2 := 52)
      { S7_Templates := "SrcType := Int" } NE_Contact(in1 := "RETAIN"."SET BOW  VCC HOLD TIME", in2 := 0)
      I_Contact( "IEC_Timer_0_DB_89".Q )
   END_RUNG wire#w5
   RUNG wire#powerrail
      { S7_Templates := "SrcType := Int" } EQ_Contact(in1 := "BUFF".PROCESS, in2 := 76)
      { S7_Templates := "SrcType := Int" } NE_Contact(in1 := "RETAIN"."SET HPHV HEAT HOLD", in2 := 0)
      I_Contact( "IEC_Timer_0_DB_83".Q )
   END_RUNG wire#w5
   RUNG wire#powerrail
      { S7_Templates := "SrcType := Int" } EQ_Contact(in1 := "BUFF".PROCESS, in2 := 56)
      { S7_Templates := "SrcType := Int" } NE_Contact(in1 := "RETAIN"."SET BOW HEAT HOLD TIME", in2 := 0)
      I_Contact( "IEC_Timer_0_DB_82".Q )
   END_RUNG wire#w5
   RUNG wire#powerrail
      { S7_Templates := "SrcType := Int" } EQ_Contact(in1 := "BUFF".PROCESS, in2 := 79)
      { S7_Templates := "SrcType := Int" } NE_Contact(in1 := "RETAIN"."SET HPHV ATS HOLD", in2 := 0)
      I_Contact( "IEC_Timer_0_DB_87".Q )
   END_RUNG wire#w5
   RUNG wire#powerrail
      { S7_Templates := "SrcType := Int" } EQ_Contact(in1 := "BUFF".PROCESS, in2 := 59)
      { S7_Templates := "SrcType := Int" } NE_Contact(in1 := "RETAIN"."SET BOW ATS HOLD", in2 := 0)
      I_Contact( "IEC_Timer_0_DB_93".Q )
   END_RUNG wire#w5
   RUNG wire#powerrail
      { S7_Templates := "SrcType := Int" } EQ_Contact(in1 := "BUFF".PROCESS, in2 := 47)
      I_Contact( "IEC_Timer_0_DB_101".Q )
   END_RUNG wire#w5
   RUNG wire#powerrail
      { S7_Templates := "SrcType := Int" } EQ_Contact(in1 := "BUFF".PROCESS, in2 := 43)
      Contact( "IEC_Timer_0_DB_97".Q )
   END_RUNG wire#w5
   RUNG wire#powerrail
      { S7_Templates := "SrcType := Int" } EQ_Contact(in1 := "BUFF".PROCESS, in2 := 45)
      Contact( "IEC_Timer_0_DB_99".Q )
   END_RUNG wire#w5
   RUNG wire#powerrail
      { S7_Templates := "SrcType := Int" } EQ_Contact(in1 := "BUFF".PROCESS, in2 := 201)
      Contact( "IEC_Timer_0_DB_170".Q )
   END_RUNG wire#w5
   RUNG wire#powerrail
      { S7_Templates := "SrcType := Int" } EQ_Contact(in1 := "BUFF".PROCESS, in2 := 251)
      Contact( "IEC_Timer_0_DB_172".Q )
   END_RUNG wire#w5
   RUNG wire#powerrail
      { S7_Templates := "SrcType := Int" } EQ_Contact(in1 := "BUFF".PROCESS, in2 := 253)
      Contact( "IEC_Timer_0_DB_175".Q )
   END_RUNG wire#w5
   RUNG wire#powerrail
      { S7_Templates := "SrcType := Int" } EQ_Contact(in1 := "BUFF".PROCESS, in2 := 255)
      Contact( "IEC_Timer_0_DB_178".Q )
   END_RUNG wire#w5
   RUNG wire#powerrail
      { S7_Templates := "SrcType := Int" } EQ_Contact(in1 := "BUFF".PROCESS, in2 := 276)
      Contact( "IEC_Timer_0_DB_180".Q )
   END_RUNG wire#w5
   RUNG wire#powerrail
      { S7_Templates := "SrcType := Int" } EQ_Contact(in1 := "BUFF".PROCESS, in2 := 278)
      Contact( "IEC_Timer_0_DB_183".Q )
   END_RUNG wire#w5
   RUNG wire#powerrail
      { S7_Templates := "SrcType := Int" } EQ_Contact(in1 := "BUFF".PROCESS, in2 := 280)
      Contact( "IEC_Timer_0_DB_186".Q )
   END_RUNG wire#w5
   // the same network as SCL:
   #_w1 := "AL STER_HOLD TIME RESET" AND NOT "pulse51";   // rising edge
   "pulse51" := "AL STER_HOLD TIME RESET";
   #_w2 := "Tag_2" AND NOT "pulse52";   // rising edge
   "pulse52" := "Tag_2";
   #_w3 := "IEC_Timer_0_DB_151".Q AND NOT "PULSE54";   // rising edge
   "PULSE54" := "IEC_Timer_0_DB_151".Q;
   #_w4 := "IEC_Timer_0_DB_152".Q AND NOT "PULSE55";   // rising edge
   "PULSE55" := "IEC_Timer_0_DB_152".Q;
   #_w5 := "IEC_Timer_0_DB_197".Q AND NOT "PULSE56";   // rising edge
   "PULSE56" := "IEC_Timer_0_DB_197".Q;
   #_w6 := "IEC_Timer_0_DB_207".Q AND NOT "PULSE66";   // rising edge
   "PULSE66" := "IEC_Timer_0_DB_207".Q;
   IF "START PV" THEN
       "SEND_PTP_DB_20"(REQ := "IEC_Counter_0_DB_2".QU OR "start process" OR "START PROCES2" OR "one shot" OR "sip_ok" OR #_w1 OR #_w2 OR #_w3 OR #_w4 OR #_w5 OR #_w6,   // SEND_PTP
                        PORT := "Local~CM_1241_(RS232)_1",
                        BUFFER := "REVAMP".L28,
                        DONE => "SEND_PTP_DB_20".DONE);
   END_IF;
   IF "START PV" THEN
       "SEND_PTP_DB_38"(REQ := "END PRINT OK" OR "sip ok1",   // SEND_PTP
                        PORT := "Local~CM_1241_(RS232)_1",
                        BUFFER := "AMEND"."PRINT PV",
                        DONE => "SEND_PTP_DB_38".DONE);
   END_IF;
   #_w7 := "vaccum ok" AND NOT "PULSE18";   // rising edge
   "PULSE18" := "vaccum ok";
   #_w8 := (("BUFF".PROCESS = 92) AND "IEC_Timer_0_DB_80".Q) OR (("BUFF".PROCESS = 492) AND "IEC_Timer_0_DB_192".Q) OR (("BUFF".PROCESS = 151) AND ("AUXILIARY"."STD VCC HOLD" <> 0) AND NOT "IEC_Timer_0_DB_95".Q) OR (("BUFF".PROCESS = 152) AND ("AUXILIARY"."STD VCC HOLD" <> 0) AND NOT "IEC_Timer_0_DB_96".Q);
   #_w9 := #_w8 AND NOT "PULSE16";   // rising edge
   "PULSE16" := #_w8;
   #_w10 := (("BUFF".PROCESS = 72) AND ("RETAIN"."SET HPHV VCC HOLD" <> 0) AND NOT "IEC_Timer_0_DB_85".Q) OR (("BUFF".PROCESS = 52) AND ("RETAIN"."SET BOW  VCC HOLD TIME" <> 0) AND NOT "IEC_Timer_0_DB_89".Q) OR (("BUFF".PROCESS = 76) AND ("RETAIN"."SET HPHV HEAT HOLD" <> 0) AND NOT "IEC_Timer_0_DB_83".Q) OR (("BUFF".PROCESS = 56) AND ("RETAIN"."SET BOW HEAT HOLD TIME" <> 0) AND NOT "IEC_Timer_0_DB_82".Q) OR (("BUFF".PROCESS = 79) AND ("RETAIN"."SET HPHV ATS HOLD" <> 0) AND NOT "IEC_Timer_0_DB_87".Q) OR (("BUFF".PROCESS = 59) AND ("RETAIN"."SET BOW ATS HOLD" <> 0) AND NOT "IEC_Timer_0_DB_93".Q) OR (("BUFF".PROCESS = 47) AND NOT "IEC_Timer_0_DB_101".Q) OR (("BUFF".PROCESS = 43) AND "IEC_Timer_0_DB_97".Q) OR (("BUFF".PROCESS = 45) AND "IEC_Timer_0_DB_99".Q) OR (("BUFF".PROCESS = 201) AND "IEC_Timer_0_DB_170".Q) OR (("BUFF".PROCESS = 251) AND "IEC_Timer_0_DB_172".Q) OR (("BUFF".PROCESS = 253) AND "IEC_Timer_0_DB_175".Q) OR (("BUFF".PROCESS = 255) AND "IEC_Timer_0_DB_178".Q) OR (("BUFF".PROCESS = 276) AND "IEC_Timer_0_DB_180".Q) OR (("BUFF".PROCESS = 278) AND "IEC_Timer_0_DB_183".Q) OR (("BUFF".PROCESS = 280) AND "IEC_Timer_0_DB_186".Q);
   #_w11 := #_w10 AND NOT "PULSE17";   // rising edge
   "PULSE17" := #_w10;
   "one shot" := #_w7 OR #_w9 OR #_w11;
END_REGION

REGION Network 16
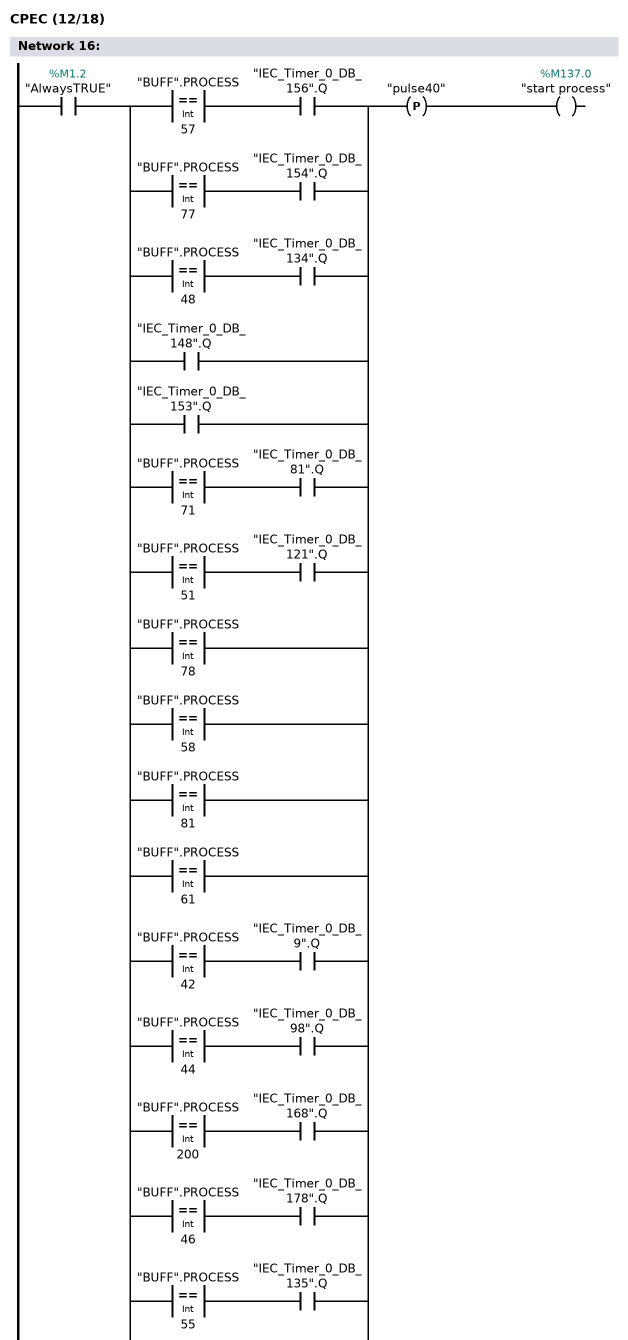
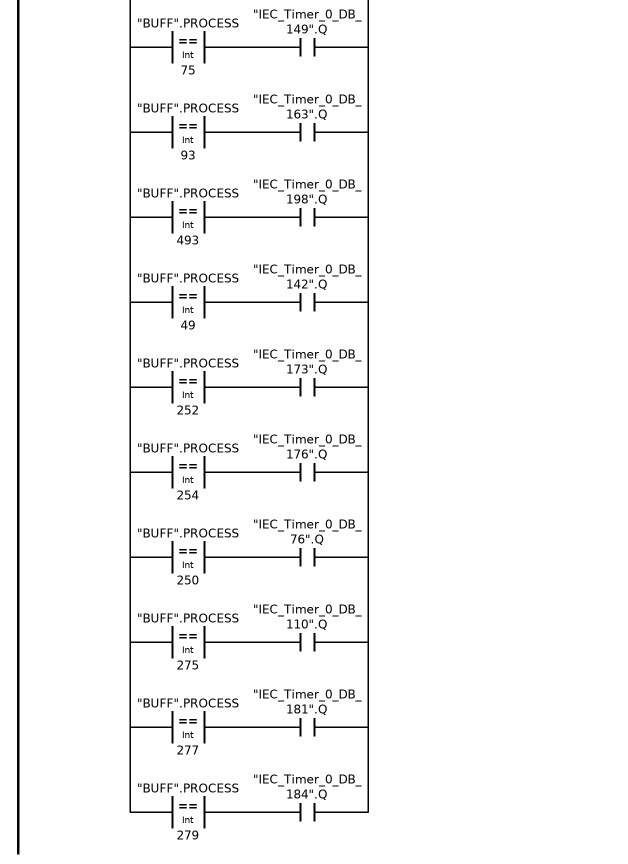
   RUNG wire#powerrail
      Contact( "AlwaysTRUE" )
      wire#w1
      { S7_Templates := "SrcType := Int" } EQ_Contact(in1 := "BUFF".PROCESS, in2 := 57)
      Contact( "IEC_Timer_0_DB_156".Q )
      wire#w2
      P_Trig( "pulse40" )
      Coil( "start process" )
   END_RUNG
   RUNG wire#w1
      { S7_Templates := "SrcType := Int" } EQ_Contact(in1 := "BUFF".PROCESS, in2 := 77)
      Contact( "IEC_Timer_0_DB_154".Q )
   END_RUNG wire#w2
   RUNG wire#w1
      { S7_Templates := "SrcType := Int" } EQ_Contact(in1 := "BUFF".PROCESS, in2 := 48)
      Contact( "IEC_Timer_0_DB_134".Q )
   END_RUNG wire#w2
   RUNG wire#w1
      Contact( "IEC_Timer_0_DB_148".Q )
   END_RUNG wire#w2
   RUNG wire#w1
      Contact( "IEC_Timer_0_DB_153".Q )
   END_RUNG wire#w2
   RUNG wire#w1
      { S7_Templates := "SrcType := Int" } EQ_Contact(in1 := "BUFF".PROCESS, in2 := 71)
      Contact( "IEC_Timer_0_DB_81".Q )
   END_RUNG wire#w2
   RUNG wire#w1
      { S7_Templates := "SrcType := Int" } EQ_Contact(in1 := "BUFF".PROCESS, in2 := 51)
      Contact( "IEC_Timer_0_DB_121".Q )
   END_RUNG wire#w2
   RUNG wire#w1
      { S7_Templates := "SrcType := Int" } EQ_Contact(in1 := "BUFF".PROCESS, in2 := 78)
   END_RUNG wire#w2
   RUNG wire#w1
      { S7_Templates := "SrcType := Int" } EQ_Contact(in1 := "BUFF".PROCESS, in2 := 58)
   END_RUNG wire#w2
   RUNG wire#w1
      { S7_Templates := "SrcType := Int" } EQ_Contact(in1 := "BUFF".PROCESS, in2 := 81)
   END_RUNG wire#w2
   RUNG wire#w1
      { S7_Templates := "SrcType := Int" } EQ_Contact(in1 := "BUFF".PROCESS, in2 := 61)
   END_RUNG wire#w2
   RUNG wire#w1
      { S7_Templates := "SrcType := Int" } EQ_Contact(in1 := "BUFF".PROCESS, in2 := 42)
      Contact( "IEC_Timer_0_DB_9".Q )
   END_RUNG wire#w2
   RUNG wire#w1
      { S7_Templates := "SrcType := Int" } EQ_Contact(in1 := "BUFF".PROCESS, in2 := 44)
      Contact( "IEC_Timer_0_DB_98".Q )
   END_RUNG wire#w2
   RUNG wire#w1
      { S7_Templates := "SrcType := Int" } EQ_Contact(in1 := "BUFF".PROCESS, in2 := 200)
      Contact( "IEC_Timer_0_DB_168".Q )
   END_RUNG wire#w2
   RUNG wire#w1
      { S7_Templates := "SrcType := Int" } EQ_Contact(in1 := "BUFF".PROCESS, in2 := 46)
      Contact( "IEC_Timer_0_DB_178".Q )
   END_RUNG wire#w2
   RUNG wire#w1
      { S7_Templates := "SrcType := Int" } EQ_Contact(in1 := "BUFF".PROCESS, in2 := 55)
      Contact( "IEC_Timer_0_DB_135".Q )
   END_RUNG wire#w2
   RUNG wire#w1
      { S7_Templates := "SrcType := Int" } EQ_Contact(in1 := "BUFF".PROCESS, in2 := 75)
      Contact( "IEC_Timer_0_DB_149".Q )
   END_RUNG wire#w2
   RUNG wire#w1
      { S7_Templates := "SrcType := Int" } EQ_Contact(in1 := "BUFF".PROCESS, in2 := 93)
      Contact( "IEC_Timer_0_DB_163".Q )
   END_RUNG wire#w2
   RUNG wire#w1
      { S7_Templates := "SrcType := Int" } EQ_Contact(in1 := "BUFF".PROCESS, in2 := 493)
      Contact( "IEC_Timer_0_DB_198".Q )
   END_RUNG wire#w2
   RUNG wire#w1
      { S7_Templates := "SrcType := Int" } EQ_Contact(in1 := "BUFF".PROCESS, in2 := 49)
      Contact( "IEC_Timer_0_DB_142".Q )
   END_RUNG wire#w2
   RUNG wire#w1
      { S7_Templates := "SrcType := Int" } EQ_Contact(in1 := "BUFF".PROCESS, in2 := 252)
      Contact( "IEC_Timer_0_DB_173".Q )
   END_RUNG wire#w2
   RUNG wire#w1
      { S7_Templates := "SrcType := Int" } EQ_Contact(in1 := "BUFF".PROCESS, in2 := 254)
      Contact( "IEC_Timer_0_DB_176".Q )
   END_RUNG wire#w2
   RUNG wire#w1
      { S7_Templates := "SrcType := Int" } EQ_Contact(in1 := "BUFF".PROCESS, in2 := 250)
      Contact( "IEC_Timer_0_DB_76".Q )
   END_RUNG wire#w2
   RUNG wire#w1
      { S7_Templates := "SrcType := Int" } EQ_Contact(in1 := "BUFF".PROCESS, in2 := 275)
      Contact( "IEC_Timer_0_DB_110".Q )
   END_RUNG wire#w2
   RUNG wire#w1
      { S7_Templates := "SrcType := Int" } EQ_Contact(in1 := "BUFF".PROCESS, in2 := 277)
      Contact( "IEC_Timer_0_DB_181".Q )
   END_RUNG wire#w2
   RUNG wire#w1
      { S7_Templates := "SrcType := Int" } EQ_Contact(in1 := "BUFF".PROCESS, in2 := 279)
      Contact( "IEC_Timer_0_DB_184".Q )
   END_RUNG wire#w2
   // the same network as SCL:
   #_w1 := "AlwaysTRUE" AND ((("BUFF".PROCESS = 57) AND "IEC_Timer_0_DB_156".Q) OR (("BUFF".PROCESS = 77) AND "IEC_Timer_0_DB_154".Q) OR (("BUFF".PROCESS = 48) AND "IEC_Timer_0_DB_134".Q) OR "IEC_Timer_0_DB_148".Q OR "IEC_Timer_0_DB_153".Q OR (("BUFF".PROCESS = 71) AND "IEC_Timer_0_DB_81".Q) OR (("BUFF".PROCESS = 51) AND "IEC_Timer_0_DB_121".Q) OR ("BUFF".PROCESS = 78) OR ("BUFF".PROCESS = 58) OR ("BUFF".PROCESS = 81) OR ("BUFF".PROCESS = 61) OR (("BUFF".PROCESS = 42) AND "IEC_Timer_0_DB_9".Q) OR (("BUFF".PROCESS = 44) AND "IEC_Timer_0_DB_98".Q) OR (("BUFF".PROCESS = 200) AND "IEC_Timer_0_DB_168".Q) OR (("BUFF".PROCESS = 46) AND "IEC_Timer_0_DB_178".Q) OR (("BUFF".PROCESS = 55) AND "IEC_Timer_0_DB_135".Q) OR (("BUFF".PROCESS = 75) AND "IEC_Timer_0_DB_149".Q) OR (("BUFF".PROCESS = 93) AND "IEC_Timer_0_DB_163".Q) OR (("BUFF".PROCESS = 493) AND "IEC_Timer_0_DB_198".Q) OR (("BUFF".PROCESS = 49) AND "IEC_Timer_0_DB_142".Q) OR (("BUFF".PROCESS = 252) AND "IEC_Timer_0_DB_173".Q) OR (("BUFF".PROCESS = 254) AND "IEC_Timer_0_DB_176".Q) OR (("BUFF".PROCESS = 250) AND "IEC_Timer_0_DB_76".Q) OR (("BUFF".PROCESS = 275) AND "IEC_Timer_0_DB_110".Q) OR (("BUFF".PROCESS = 277) AND "IEC_Timer_0_DB_181".Q) OR (("BUFF".PROCESS = 279) AND "IEC_Timer_0_DB_184".Q));
   #_w2 := #_w1 AND NOT "pulse40";   // rising edge
   "pulse40" := #_w1;
   "start process" := #_w2;
END_REGION

REGION Network 17
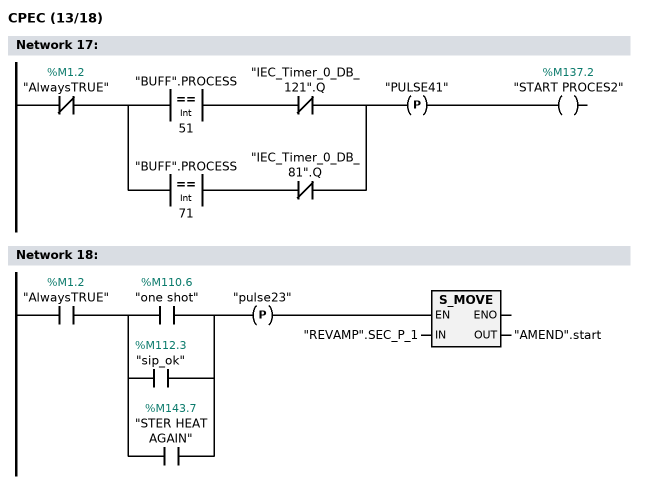
   RUNG wire#powerrail
      I_Contact( "AlwaysTRUE" )
      wire#w1
      { S7_Templates := "SrcType := Int" } EQ_Contact(in1 := "BUFF".PROCESS, in2 := 51)
      I_Contact( "IEC_Timer_0_DB_121".Q )
      wire#w2
      P_Trig( "PULSE41" )
      Coil( "START PROCES2" )
   END_RUNG
   RUNG wire#w1
      { S7_Templates := "SrcType := Int" } EQ_Contact(in1 := "BUFF".PROCESS, in2 := 71)
      I_Contact( "IEC_Timer_0_DB_81".Q )
   END_RUNG wire#w2
   // the same network as SCL:
   #_w1 := NOT "AlwaysTRUE" AND ((("BUFF".PROCESS = 51) AND NOT "IEC_Timer_0_DB_121".Q) OR (("BUFF".PROCESS = 71) AND NOT "IEC_Timer_0_DB_81".Q));
   #_w2 := #_w1 AND NOT "PULSE41";   // rising edge
   "PULSE41" := #_w1;
   "START PROCES2" := #_w2;
END_REGION

REGION Network 18
   RUNG wire#powerrail
      Contact( "AlwaysTRUE" )
      wire#w1
      Contact( "one shot" )
      wire#w2
      P_Trig( "pulse23" )
      S_Move(in := "REVAMP".SEC_P_1, out => "AMEND".start)
   END_RUNG
   RUNG wire#w1
      Contact( "sip_ok" )
   END_RUNG wire#w2
   RUNG wire#w1
      Contact( "STER HEAT AGAIN" )
   END_RUNG wire#w2
   // the same network as SCL:
   #_w1 := "AlwaysTRUE" AND ("one shot" OR "sip_ok" OR "STER HEAT AGAIN");
   #_w2 := #_w1 AND NOT "pulse23";   // rising edge
   "pulse23" := #_w1;
   IF #_w2 THEN "AMEND".start := "REVAMP".SEC_P_1; END_IF;
END_REGION

REGION Network 19
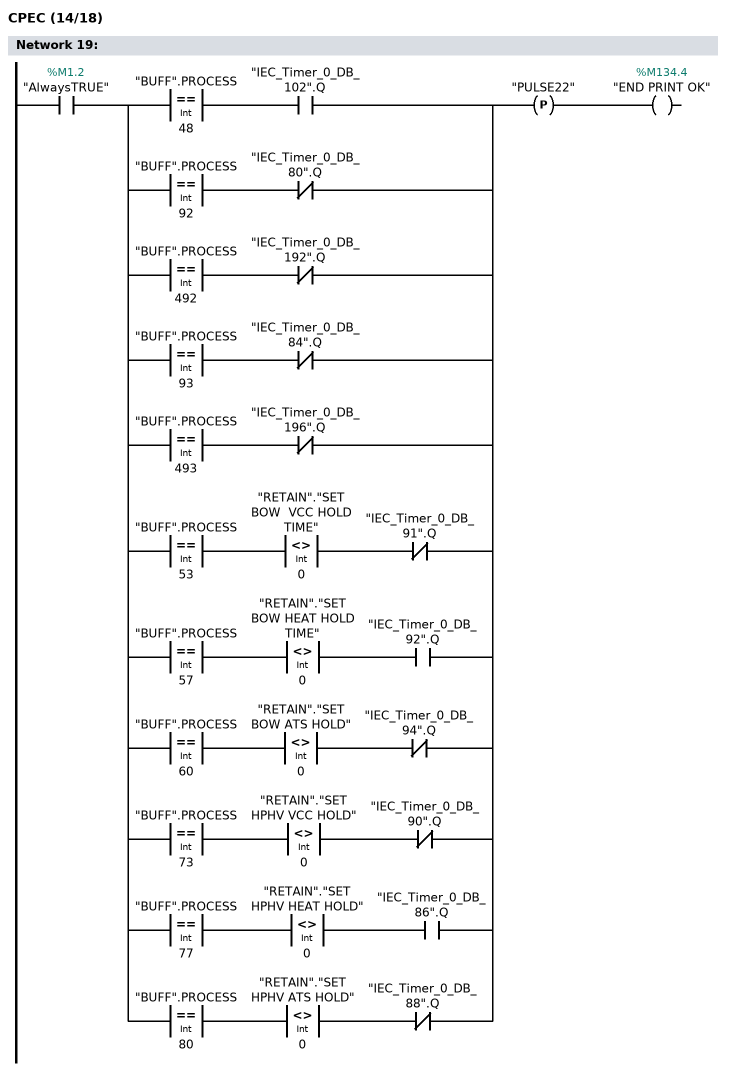
   RUNG wire#powerrail
      Contact( "AlwaysTRUE" )
      wire#w1
      { S7_Templates := "SrcType := Int" } EQ_Contact(in1 := "BUFF".PROCESS, in2 := 48)
      Contact( "IEC_Timer_0_DB_102".Q )
      wire#w2
      P_Trig( "PULSE22" )
      Coil( "END PRINT OK" )
   END_RUNG
   RUNG wire#w1
      { S7_Templates := "SrcType := Int" } EQ_Contact(in1 := "BUFF".PROCESS, in2 := 92)
      I_Contact( "IEC_Timer_0_DB_80".Q )
   END_RUNG wire#w2
   RUNG wire#w1
      { S7_Templates := "SrcType := Int" } EQ_Contact(in1 := "BUFF".PROCESS, in2 := 492)
      I_Contact( "IEC_Timer_0_DB_192".Q )
   END_RUNG wire#w2
   RUNG wire#w1
      { S7_Templates := "SrcType := Int" } EQ_Contact(in1 := "BUFF".PROCESS, in2 := 93)
      I_Contact( "IEC_Timer_0_DB_84".Q )
   END_RUNG wire#w2
   RUNG wire#w1
      { S7_Templates := "SrcType := Int" } EQ_Contact(in1 := "BUFF".PROCESS, in2 := 493)
      I_Contact( "IEC_Timer_0_DB_196".Q )
   END_RUNG wire#w2
   RUNG wire#w1
      { S7_Templates := "SrcType := Int" } EQ_Contact(in1 := "BUFF".PROCESS, in2 := 53)
      { S7_Templates := "SrcType := Int" } NE_Contact(in1 := "RETAIN"."SET BOW  VCC HOLD TIME", in2 := 0)
      I_Contact( "IEC_Timer_0_DB_91".Q )
   END_RUNG wire#w2
   RUNG wire#w1
      { S7_Templates := "SrcType := Int" } EQ_Contact(in1 := "BUFF".PROCESS, in2 := 57)
      { S7_Templates := "SrcType := Int" } NE_Contact(in1 := "RETAIN"."SET BOW HEAT HOLD TIME", in2 := 0)
      Contact( "IEC_Timer_0_DB_92".Q )
   END_RUNG wire#w2
   RUNG wire#w1
      { S7_Templates := "SrcType := Int" } EQ_Contact(in1 := "BUFF".PROCESS, in2 := 60)
      { S7_Templates := "SrcType := Int" } NE_Contact(in1 := "RETAIN"."SET BOW ATS HOLD", in2 := 0)
      I_Contact( "IEC_Timer_0_DB_94".Q )
   END_RUNG wire#w2
   RUNG wire#w1
      { S7_Templates := "SrcType := Int" } EQ_Contact(in1 := "BUFF".PROCESS, in2 := 73)
      { S7_Templates := "SrcType := Int" } NE_Contact(in1 := "RETAIN"."SET HPHV VCC HOLD", in2 := 0)
      I_Contact( "IEC_Timer_0_DB_90".Q )
   END_RUNG wire#w2
   RUNG wire#w1
      { S7_Templates := "SrcType := Int" } EQ_Contact(in1 := "BUFF".PROCESS, in2 := 77)
      { S7_Templates := "SrcType := Int" } NE_Contact(in1 := "RETAIN"."SET HPHV HEAT HOLD", in2 := 0)
      Contact( "IEC_Timer_0_DB_86".Q )
   END_RUNG wire#w2
   RUNG wire#w1
      { S7_Templates := "SrcType := Int" } EQ_Contact(in1 := "BUFF".PROCESS, in2 := 80)
      { S7_Templates := "SrcType := Int" } NE_Contact(in1 := "RETAIN"."SET HPHV ATS HOLD", in2 := 0)
      I_Contact( "IEC_Timer_0_DB_88".Q )
   END_RUNG wire#w2
   // the same network as SCL:
   #_w1 := "AlwaysTRUE" AND ((("BUFF".PROCESS = 48) AND "IEC_Timer_0_DB_102".Q) OR (("BUFF".PROCESS = 92) AND NOT "IEC_Timer_0_DB_80".Q) OR (("BUFF".PROCESS = 492) AND NOT "IEC_Timer_0_DB_192".Q) OR (("BUFF".PROCESS = 93) AND NOT "IEC_Timer_0_DB_84".Q) OR (("BUFF".PROCESS = 493) AND NOT "IEC_Timer_0_DB_196".Q) OR (("BUFF".PROCESS = 53) AND ("RETAIN"."SET BOW  VCC HOLD TIME" <> 0) AND NOT "IEC_Timer_0_DB_91".Q) OR (("BUFF".PROCESS = 57) AND ("RETAIN"."SET BOW HEAT HOLD TIME" <> 0) AND "IEC_Timer_0_DB_92".Q) OR (("BUFF".PROCESS = 60) AND ("RETAIN"."SET BOW ATS HOLD" <> 0) AND NOT "IEC_Timer_0_DB_94".Q) OR (("BUFF".PROCESS = 73) AND ("RETAIN"."SET HPHV VCC HOLD" <> 0) AND NOT "IEC_Timer_0_DB_90".Q) OR (("BUFF".PROCESS = 77) AND ("RETAIN"."SET HPHV HEAT HOLD" <> 0) AND "IEC_Timer_0_DB_86".Q) OR (("BUFF".PROCESS = 80) AND ("RETAIN"."SET HPHV ATS HOLD" <> 0) AND NOT "IEC_Timer_0_DB_88".Q));
   #_w2 := #_w1 AND NOT "PULSE22";   // rising edge
   "PULSE22" := #_w1;
   "END PRINT OK" := #_w2;
END_REGION

REGION Network 20
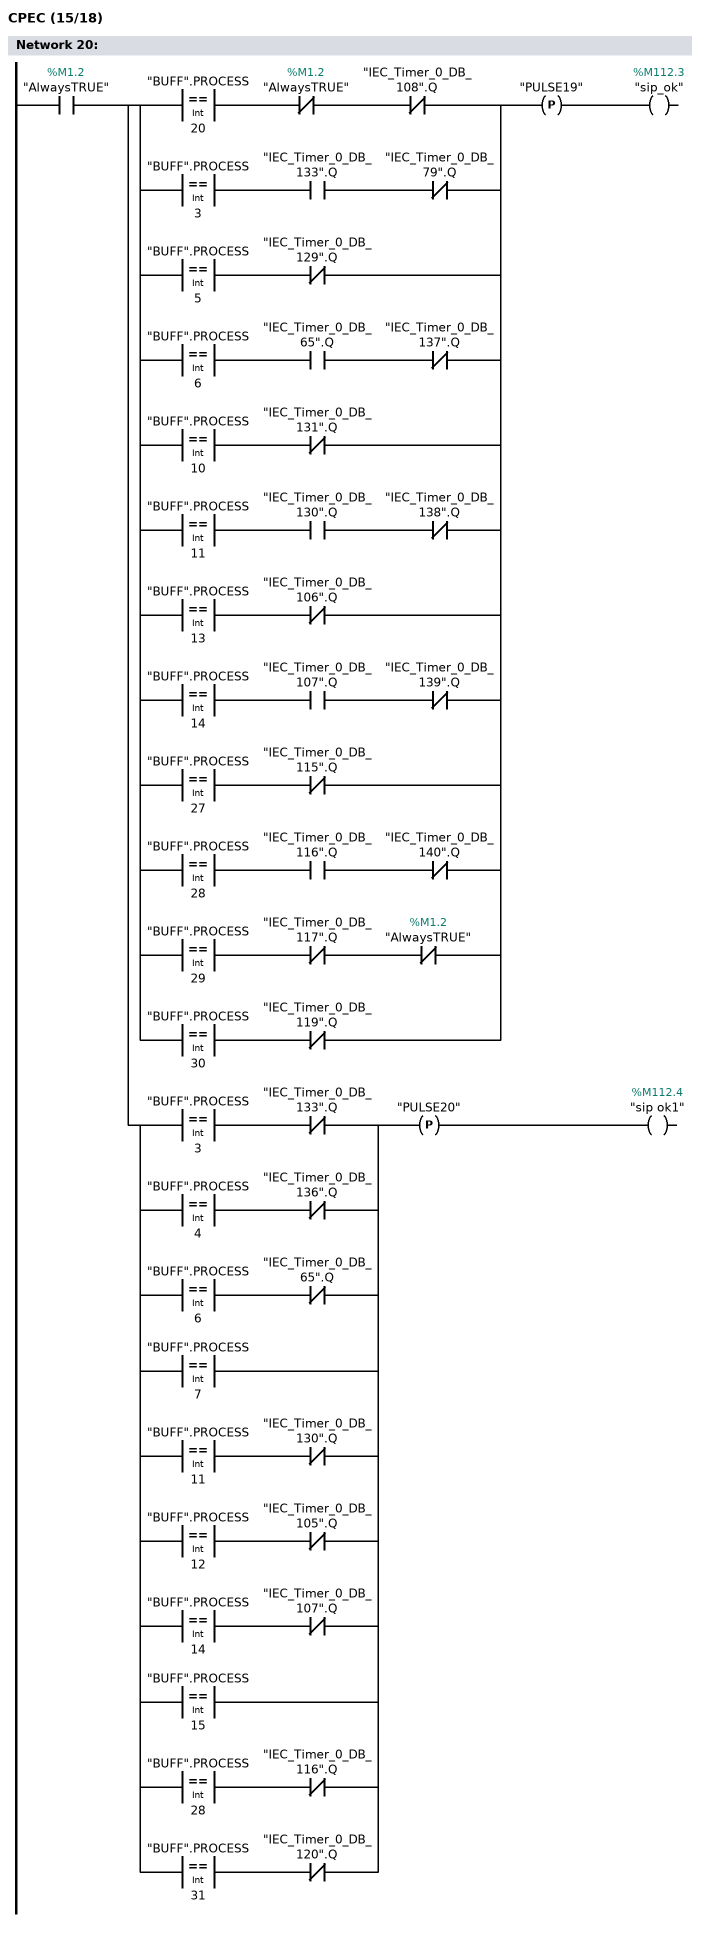
   RUNG wire#powerrail
      Contact( "AlwaysTRUE" )
      wire#w1
      { S7_Templates := "SrcType := Int" } EQ_Contact(in1 := "BUFF".PROCESS, in2 := 20)
      I_Contact( "AlwaysTRUE" )
      I_Contact( "IEC_Timer_0_DB_108".Q )
      wire#w2
      P_Trig( "PULSE19" )
      Coil( "sip_ok" )
   END_RUNG
   RUNG wire#w1
      { S7_Templates := "SrcType := Int" } EQ_Contact(in1 := "BUFF".PROCESS, in2 := 3)
      Contact( "IEC_Timer_0_DB_133".Q )
      I_Contact( "IEC_Timer_0_DB_79".Q )
   END_RUNG wire#w2
   RUNG wire#w1
      { S7_Templates := "SrcType := Int" } EQ_Contact(in1 := "BUFF".PROCESS, in2 := 5)
      I_Contact( "IEC_Timer_0_DB_129".Q )
   END_RUNG wire#w2
   RUNG wire#w1
      { S7_Templates := "SrcType := Int" } EQ_Contact(in1 := "BUFF".PROCESS, in2 := 6)
      Contact( "IEC_Timer_0_DB_65".Q )
      I_Contact( "IEC_Timer_0_DB_137".Q )
   END_RUNG wire#w2
   RUNG wire#w1
      { S7_Templates := "SrcType := Int" } EQ_Contact(in1 := "BUFF".PROCESS, in2 := 10)
      I_Contact( "IEC_Timer_0_DB_131".Q )
   END_RUNG wire#w2
   RUNG wire#w1
      { S7_Templates := "SrcType := Int" } EQ_Contact(in1 := "BUFF".PROCESS, in2 := 11)
      Contact( "IEC_Timer_0_DB_130".Q )
      I_Contact( "IEC_Timer_0_DB_138".Q )
   END_RUNG wire#w2
   RUNG wire#w1
      { S7_Templates := "SrcType := Int" } EQ_Contact(in1 := "BUFF".PROCESS, in2 := 13)
      I_Contact( "IEC_Timer_0_DB_106".Q )
   END_RUNG wire#w2
   RUNG wire#w1
      { S7_Templates := "SrcType := Int" } EQ_Contact(in1 := "BUFF".PROCESS, in2 := 14)
      Contact( "IEC_Timer_0_DB_107".Q )
      I_Contact( "IEC_Timer_0_DB_139".Q )
   END_RUNG wire#w2
   RUNG wire#w1
      { S7_Templates := "SrcType := Int" } EQ_Contact(in1 := "BUFF".PROCESS, in2 := 27)
      I_Contact( "IEC_Timer_0_DB_115".Q )
   END_RUNG wire#w2
   RUNG wire#w1
      { S7_Templates := "SrcType := Int" } EQ_Contact(in1 := "BUFF".PROCESS, in2 := 28)
      Contact( "IEC_Timer_0_DB_116".Q )
      I_Contact( "IEC_Timer_0_DB_140".Q )
   END_RUNG wire#w2
   RUNG wire#w1
      { S7_Templates := "SrcType := Int" } EQ_Contact(in1 := "BUFF".PROCESS, in2 := 29)
      I_Contact( "IEC_Timer_0_DB_117".Q )
      I_Contact( "AlwaysTRUE" )
   END_RUNG wire#w2
   RUNG wire#w1
      { S7_Templates := "SrcType := Int" } EQ_Contact(in1 := "BUFF".PROCESS, in2 := 30)
      I_Contact( "IEC_Timer_0_DB_119".Q )
   END_RUNG wire#w2
   RUNG wire#w1
      { S7_Templates := "SrcType := Int" } EQ_Contact(in1 := "BUFF".PROCESS, in2 := 3)
      I_Contact( "IEC_Timer_0_DB_133".Q )
      wire#w3
      P_Trig( "PULSE20" )
      Coil( "sip ok1" )
   END_RUNG
   RUNG wire#w1
      { S7_Templates := "SrcType := Int" } EQ_Contact(in1 := "BUFF".PROCESS, in2 := 4)
      I_Contact( "IEC_Timer_0_DB_136".Q )
   END_RUNG wire#w3
   RUNG wire#w1
      { S7_Templates := "SrcType := Int" } EQ_Contact(in1 := "BUFF".PROCESS, in2 := 6)
      I_Contact( "IEC_Timer_0_DB_65".Q )
   END_RUNG wire#w3
   RUNG wire#w1
      { S7_Templates := "SrcType := Int" } EQ_Contact(in1 := "BUFF".PROCESS, in2 := 7)
   END_RUNG wire#w3
   RUNG wire#w1
      { S7_Templates := "SrcType := Int" } EQ_Contact(in1 := "BUFF".PROCESS, in2 := 11)
      I_Contact( "IEC_Timer_0_DB_130".Q )
   END_RUNG wire#w3
   RUNG wire#w1
      { S7_Templates := "SrcType := Int" } EQ_Contact(in1 := "BUFF".PROCESS, in2 := 12)
      I_Contact( "IEC_Timer_0_DB_105".Q )
   END_RUNG wire#w3
   RUNG wire#w1
      { S7_Templates := "SrcType := Int" } EQ_Contact(in1 := "BUFF".PROCESS, in2 := 14)
      I_Contact( "IEC_Timer_0_DB_107".Q )
   END_RUNG wire#w3
   RUNG wire#w1
      { S7_Templates := "SrcType := Int" } EQ_Contact(in1 := "BUFF".PROCESS, in2 := 15)
   END_RUNG wire#w3
   RUNG wire#w1
      { S7_Templates := "SrcType := Int" } EQ_Contact(in1 := "BUFF".PROCESS, in2 := 28)
      I_Contact( "IEC_Timer_0_DB_116".Q )
   END_RUNG wire#w3
   RUNG wire#w1
      { S7_Templates := "SrcType := Int" } EQ_Contact(in1 := "BUFF".PROCESS, in2 := 31)
      I_Contact( "IEC_Timer_0_DB_120".Q )
   END_RUNG wire#w3
   // the same network as SCL:
   #_w1 := "AlwaysTRUE" AND ((("BUFF".PROCESS = 20) AND NOT "AlwaysTRUE" AND NOT "IEC_Timer_0_DB_108".Q) OR (("BUFF".PROCESS = 3) AND "IEC_Timer_0_DB_133".Q AND NOT "IEC_Timer_0_DB_79".Q) OR (("BUFF".PROCESS = 5) AND NOT "IEC_Timer_0_DB_129".Q) OR (("BUFF".PROCESS = 6) AND "IEC_Timer_0_DB_65".Q AND NOT "IEC_Timer_0_DB_137".Q) OR (("BUFF".PROCESS = 10) AND NOT "IEC_Timer_0_DB_131".Q) OR (("BUFF".PROCESS = 11) AND "IEC_Timer_0_DB_130".Q AND NOT "IEC_Timer_0_DB_138".Q) OR (("BUFF".PROCESS = 13) AND NOT "IEC_Timer_0_DB_106".Q) OR (("BUFF".PROCESS = 14) AND "IEC_Timer_0_DB_107".Q AND NOT "IEC_Timer_0_DB_139".Q) OR (("BUFF".PROCESS = 27) AND NOT "IEC_Timer_0_DB_115".Q) OR (("BUFF".PROCESS = 28) AND "IEC_Timer_0_DB_116".Q AND NOT "IEC_Timer_0_DB_140".Q) OR (("BUFF".PROCESS = 29) AND NOT "IEC_Timer_0_DB_117".Q AND NOT "AlwaysTRUE") OR (("BUFF".PROCESS = 30) AND NOT "IEC_Timer_0_DB_119".Q));
   #_w2 := #_w1 AND NOT "PULSE19";   // rising edge
   "PULSE19" := #_w1;
   "sip_ok" := #_w2;
   #_w3 := "AlwaysTRUE" AND ((("BUFF".PROCESS = 3) AND NOT "IEC_Timer_0_DB_133".Q) OR (("BUFF".PROCESS = 4) AND NOT "IEC_Timer_0_DB_136".Q) OR (("BUFF".PROCESS = 6) AND NOT "IEC_Timer_0_DB_65".Q) OR ("BUFF".PROCESS = 7) OR (("BUFF".PROCESS = 11) AND NOT "IEC_Timer_0_DB_130".Q) OR (("BUFF".PROCESS = 12) AND NOT "IEC_Timer_0_DB_105".Q) OR (("BUFF".PROCESS = 14) AND NOT "IEC_Timer_0_DB_107".Q) OR ("BUFF".PROCESS = 15) OR (("BUFF".PROCESS = 28) AND NOT "IEC_Timer_0_DB_116".Q) OR (("BUFF".PROCESS = 31) AND NOT "IEC_Timer_0_DB_120".Q));
   #_w4 := #_w3 AND NOT "PULSE20";   // rising edge
   "PULSE20" := #_w3;
   "sip ok1" := #_w4;
END_REGION

REGION Network 21
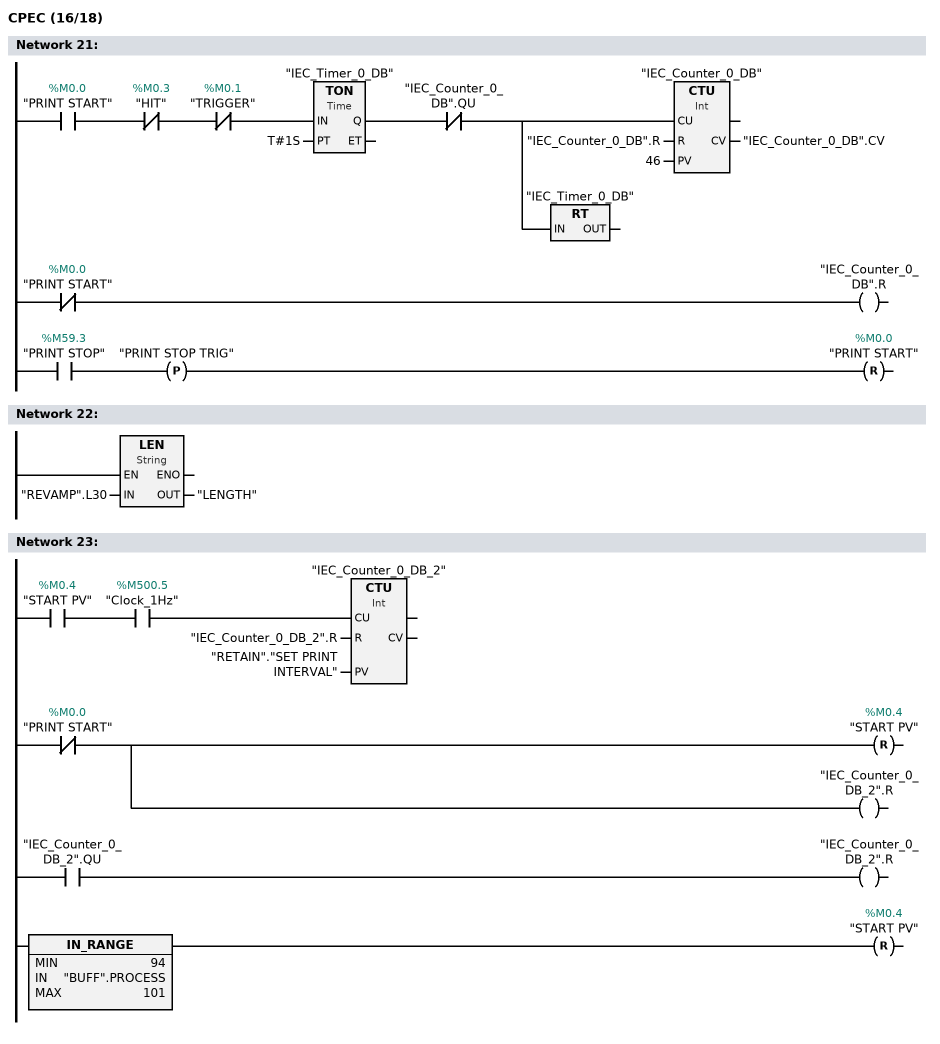
   RUNG wire#powerrail
      Contact( "PRINT START" )
      I_Contact( "HIT" )
      I_Contact( "TRIGGER" )
      { S7_Templates := "time_type := Time" } "IEC_Timer_0_DB".TON(pt := T#1S, et =>)
      I_Contact( "IEC_Counter_0_DB".QU )
      wire#w1
      { S7_Templates := "value_type := Int" } "IEC_Counter_0_DB".CTU(r := "IEC_Counter_0_DB".R, pv := 46, cv => "IEC_Counter_0_DB".CV)
   END_RUNG
   RUNG wire#w1
      RT_Coil( "IEC_Timer_0_DB" )
   END_RUNG
   RUNG wire#powerrail
      I_Contact( "PRINT START" )
      Coil( "IEC_Counter_0_DB".R )
   END_RUNG
   RUNG wire#powerrail
      Contact( "PRINT STOP" )
      P_Trig( "PRINT STOP TRIG" )
      R_Coil( "PRINT START" )
   END_RUNG
   // the same network as SCL:
   "IEC_Timer_0_DB".TON(IN := "PRINT START" AND NOT "HIT" AND NOT "TRIGGER", PT := T#1S);
   #_w1 := "IEC_Timer_0_DB".Q AND NOT "IEC_Counter_0_DB".QU;
   "IEC_Counter_0_DB".CTU(CU := #_w1, R := "IEC_Counter_0_DB".R, PV := 46, CV => "IEC_Counter_0_DB".CV);
   IF #_w1 THEN RESET_TIMER("IEC_Timer_0_DB"); END_IF;
   "IEC_Counter_0_DB".R := NOT "PRINT START";
   #_w2 := "PRINT STOP" AND NOT "PRINT STOP TRIG";   // rising edge
   "PRINT STOP TRIG" := "PRINT STOP";
   IF #_w2 THEN "PRINT START" := FALSE; END_IF;
END_REGION

REGION Network 22
   RUNG wire#powerrail
      { S7_Templates := "[str_type := String, return_type := Int]" } LEN(IN := "REVAMP".L30, OUT => "LENGTH")
   END_RUNG
   // the same network as SCL:
   LEN(IN := "REVAMP".L30, OUT => "LENGTH");
END_REGION

REGION Network 23
   RUNG wire#powerrail
      Contact( "START PV" )
      Contact( "Clock_1Hz" )
      { S7_Templates := "value_type := Int" } "IEC_Counter_0_DB_2".CTU(r := "IEC_Counter_0_DB_2".R, pv := "RETAIN"."SET PRINT INTERVAL", cv =>)
   END_RUNG
   RUNG wire#powerrail
      I_Contact( "PRINT START" )
      wire#w1
      R_Coil( "START PV" )
   END_RUNG
   RUNG wire#w1
      Coil( "IEC_Counter_0_DB_2".R )
   END_RUNG
   RUNG wire#powerrail
      Contact( "IEC_Counter_0_DB_2".QU )
      Coil( "IEC_Counter_0_DB_2".R )
   END_RUNG
   RUNG wire#powerrail
      { S7_Templates := "SrcType := Int" } InRange(min := 94, in := "BUFF".PROCESS, max := 101)
      R_Coil( "START PV" )
   END_RUNG
   // the same network as SCL:
   "IEC_Counter_0_DB_2".CTU(CU := "START PV" AND "Clock_1Hz",
                           R := "IEC_Counter_0_DB_2".R,
                           PV := "RETAIN"."SET PRINT INTERVAL");
   IF NOT "PRINT START" THEN "START PV" := FALSE; END_IF;
   "IEC_Counter_0_DB_2".R := NOT "PRINT START";
   "IEC_Counter_0_DB_2".R := "IEC_Counter_0_DB_2".QU;
   IF (94 <= "BUFF".PROCESS) AND ("BUFF".PROCESS <= 101) THEN "START PV" := FALSE; END_IF;
END_REGION

REGION Network 24
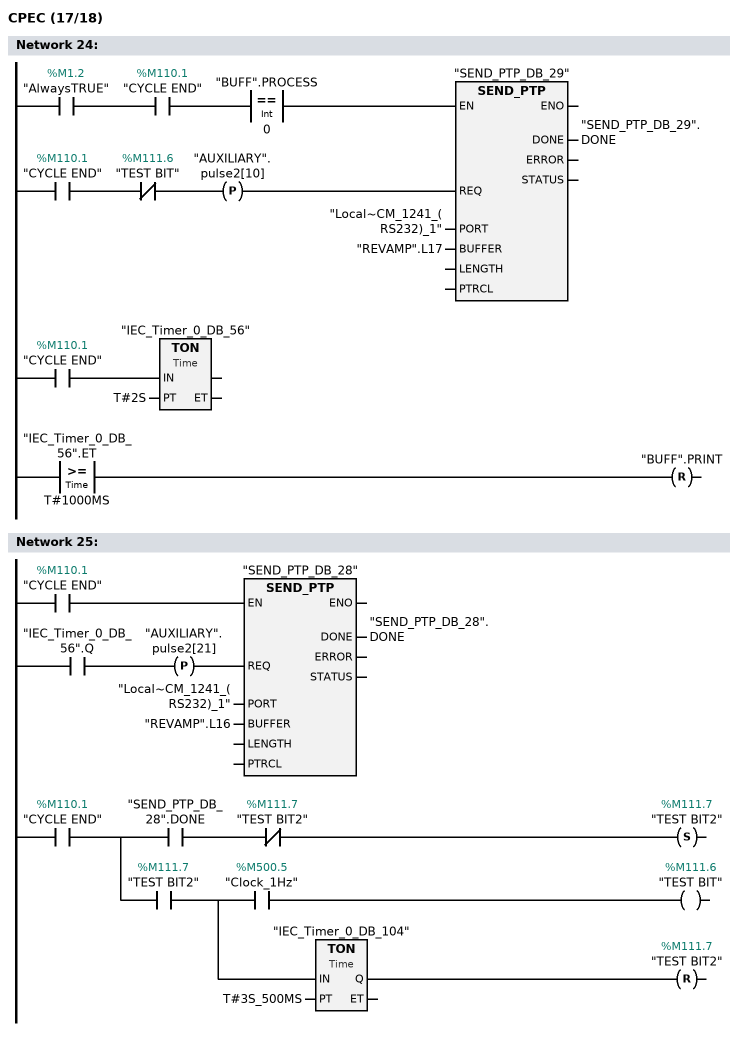
   RUNG wire#powerrail
      Contact( "AlwaysTRUE" )
      Contact( "CYCLE END" )
      { S7_Templates := "SrcType := Int" } EQ_Contact(in1 := "BUFF".PROCESS, in2 := 0)
      "SEND_PTP_DB_29".SEND_PTP(REQ := wire#w1, PORT := "Local~CM_1241_(RS232)_1", BUFFER := "REVAMP".L17, LENGTH :=, PTRCL :=, DONE => "SEND_PTP_DB_29".DONE, ERROR =>, STATUS =>)
   END_RUNG
   RUNG wire#powerrail
      Contact( "CYCLE END" )
      I_Contact( "TEST BIT" )
      P_Trig( "AUXILIARY".pulse2[10] )
   END_RUNG wire#w1
   RUNG wire#powerrail
      Contact( "CYCLE END" )
      { S7_Templates := "time_type := Time" } "IEC_Timer_0_DB_56".TON(pt := T#2S, et =>)
   END_RUNG
   RUNG wire#powerrail
      { S7_Templates := "SrcType := Time" } GE_Contact(in1 := "IEC_Timer_0_DB_56".ET, in2 := T#1000MS)
      R_Coil( "BUFF".PRINT )
   END_RUNG
   // the same network as SCL:
   #_w1 := "CYCLE END" AND NOT "TEST BIT";
   #_w2 := #_w1 AND NOT "AUXILIARY".pulse2[10];   // rising edge
   "AUXILIARY".pulse2[10] := #_w1;
   IF "AlwaysTRUE" AND "CYCLE END" AND ("BUFF".PROCESS = 0) THEN
       "SEND_PTP_DB_29"(REQ := #_w2,   // SEND_PTP
                        PORT := "Local~CM_1241_(RS232)_1",
                        BUFFER := "REVAMP".L17,
                        DONE => "SEND_PTP_DB_29".DONE);
   END_IF;
   "IEC_Timer_0_DB_56".TON(IN := "CYCLE END", PT := T#2S);
   IF "IEC_Timer_0_DB_56".ET >= T#1000MS THEN "BUFF".PRINT := FALSE; END_IF;
END_REGION

REGION Network 25
   RUNG wire#powerrail
      Contact( "CYCLE END" )
      "SEND_PTP_DB_28".SEND_PTP(REQ := wire#w1, PORT := "Local~CM_1241_(RS232)_1", BUFFER := "REVAMP".L16, LENGTH :=, PTRCL :=, DONE => "SEND_PTP_DB_28".DONE, ERROR =>, STATUS =>)
   END_RUNG
   RUNG wire#powerrail
      Contact( "IEC_Timer_0_DB_56".Q )
      P_Trig( "AUXILIARY".pulse2[21] )
   END_RUNG wire#w1
   RUNG wire#powerrail
      Contact( "CYCLE END" )
      wire#w2
      Contact( "SEND_PTP_DB_28".DONE )
      I_Contact( "TEST BIT2" )
      S_Coil( "TEST BIT2" )
   END_RUNG
   RUNG wire#w2
      Contact( "TEST BIT2" )
      wire#w3
      Contact( "Clock_1Hz" )
      Coil( "TEST BIT" )
   END_RUNG
   RUNG wire#w3
      { S7_Templates := "time_type := Time" } "IEC_Timer_0_DB_104".TON(pt := T#3S_500MS, et =>)
      R_Coil( "TEST BIT2" )
   END_RUNG
   // the same network as SCL:
   #_w1 := "IEC_Timer_0_DB_56".Q AND NOT "AUXILIARY".pulse2[21];   // rising edge
   "AUXILIARY".pulse2[21] := "IEC_Timer_0_DB_56".Q;
   IF "CYCLE END" THEN
       "SEND_PTP_DB_28"(REQ := #_w1,   // SEND_PTP
                        PORT := "Local~CM_1241_(RS232)_1",
                        BUFFER := "REVAMP".L16,
                        DONE => "SEND_PTP_DB_28".DONE);
   END_IF;
   IF "CYCLE END" AND "SEND_PTP_DB_28".DONE AND NOT "TEST BIT2" THEN "TEST BIT2" := TRUE; END_IF;
   #_w2 := "CYCLE END" AND "TEST BIT2";
   "TEST BIT" := #_w2 AND "Clock_1Hz";
   "IEC_Timer_0_DB_104".TON(IN := #_w2, PT := T#3S_500MS);
   IF "IEC_Timer_0_DB_104".Q THEN "TEST BIT2" := FALSE; END_IF;
END_REGION

REGION Network 26
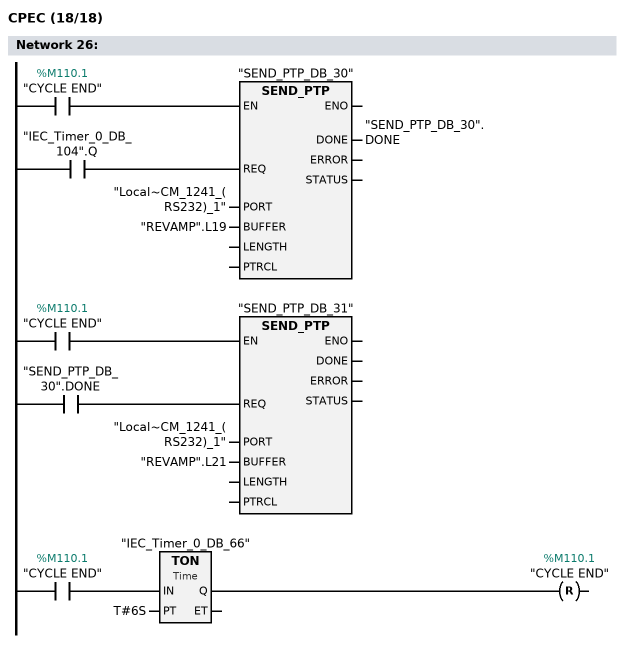
   RUNG wire#powerrail
      Contact( "CYCLE END" )
      "SEND_PTP_DB_30".SEND_PTP(REQ := wire#w1, PORT := "Local~CM_1241_(RS232)_1", BUFFER := "REVAMP".L19, LENGTH :=, PTRCL :=, DONE => "SEND_PTP_DB_30".DONE, ERROR =>, STATUS =>)
   END_RUNG
   RUNG wire#powerrail
      Contact( "IEC_Timer_0_DB_104".Q )
   END_RUNG wire#w1
   RUNG wire#powerrail
      Contact( "CYCLE END" )
      "SEND_PTP_DB_31".SEND_PTP(REQ := wire#w2, PORT := "Local~CM_1241_(RS232)_1", BUFFER := "REVAMP".L21, LENGTH :=, PTRCL :=, DONE =>, ERROR =>, STATUS =>)
   END_RUNG
   RUNG wire#powerrail
      Contact( "SEND_PTP_DB_30".DONE )
   END_RUNG wire#w2
   RUNG wire#powerrail
      Contact( "CYCLE END" )
      { S7_Templates := "time_type := Time" } "IEC_Timer_0_DB_66".TON(pt := T#6S, et =>)
      R_Coil( "CYCLE END" )
   END_RUNG
   // the same network as SCL:
   IF "CYCLE END" THEN
       "SEND_PTP_DB_30"(REQ := "IEC_Timer_0_DB_104".Q,   // SEND_PTP
                        PORT := "Local~CM_1241_(RS232)_1",
                        BUFFER := "REVAMP".L19,
                        DONE => "SEND_PTP_DB_30".DONE);
   END_IF;
   IF "CYCLE END" THEN
       "SEND_PTP_DB_31"(REQ := "SEND_PTP_DB_30".DONE, PORT := "Local~CM_1241_(RS232)_1", BUFFER := "REVAMP".L21);   // SEND_PTP
   END_IF;
   "IEC_Timer_0_DB_66".TON(IN := "CYCLE END", PT := T#6S);
   IF "IEC_Timer_0_DB_66".Q THEN "CYCLE END" := FALSE; END_IF;
END_REGION
END_FUNCTION

FUNCTION "HPHV" : Void   // FC11, LAD
{ S7_Optimized_Access := 'TRUE' }
// stored: SetENOAutomatically false
   VAR_TEMP
      "HOLD START" : Bool;
   END_VAR
   VAR_TEMP   // added for the SCL form of the ladder/FBD networks
      _w1 : Bool;
      _w2 : Bool;
      _w3 : Bool;
      _w4 : Bool;
   END_VAR
BEGIN

REGION Network 1
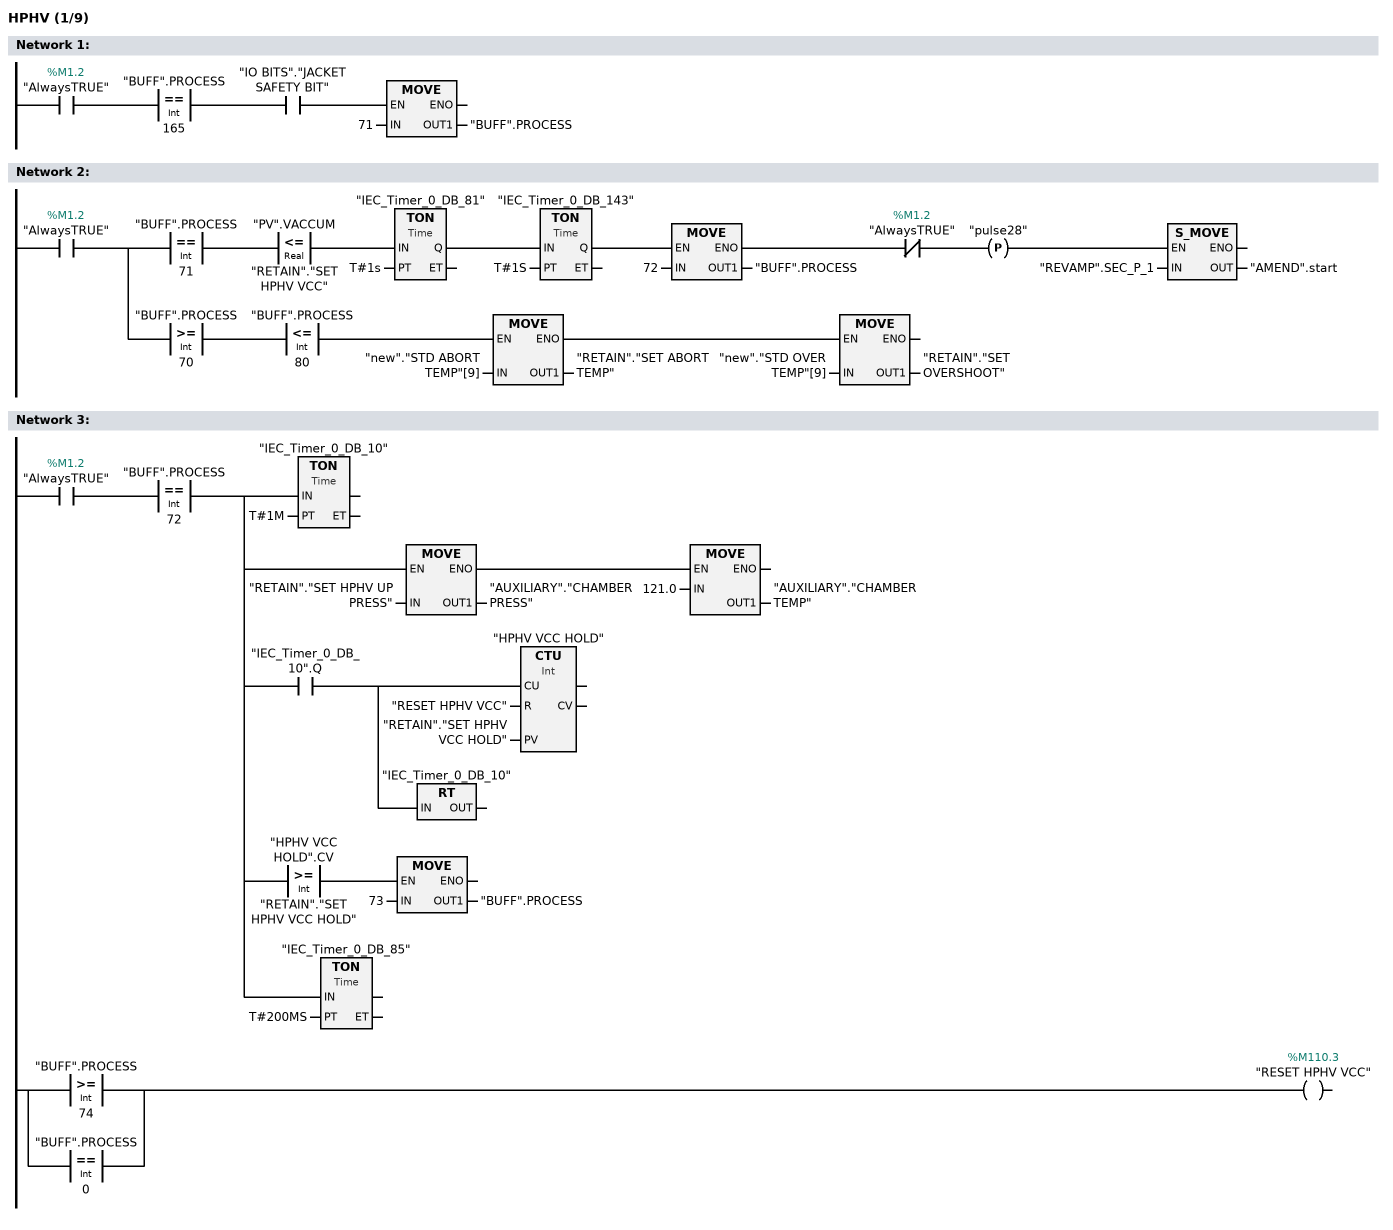
   RUNG wire#powerrail
      Contact( "AlwaysTRUE" )
      { S7_Templates := "SrcType := Int" } EQ_Contact(in1 := "BUFF".PROCESS, in2 := 165)
      Contact( "IO BITS"."JACKET SAFETY BIT" )
      Move(in := 71, out1 => "BUFF".PROCESS)
   END_RUNG
   // the same network as SCL:
   IF "AlwaysTRUE" AND ("BUFF".PROCESS = 165) AND "IO BITS"."JACKET SAFETY BIT" THEN
       "BUFF".PROCESS := 71;
   END_IF;
END_REGION

REGION Network 2
   RUNG wire#powerrail
      Contact( "AlwaysTRUE" )
      wire#w1
      { S7_Templates := "SrcType := Int" } EQ_Contact(in1 := "BUFF".PROCESS, in2 := 71)
      { S7_Templates := "SrcType := Real" } LE_Contact(in1 := "PV".VACCUM, in2 := "RETAIN"."SET HPHV VCC")
      { S7_Templates := "time_type := Time" } "IEC_Timer_0_DB_81".TON(pt := T#1s, et =>)
      { S7_Templates := "time_type := Time" } "IEC_Timer_0_DB_143".TON(pt := T#1S, et =>)
      Move(in := 72, out1 => "BUFF".PROCESS)
      I_Contact( "AlwaysTRUE" )
      P_Trig( "pulse28" )
      S_Move(in := "REVAMP".SEC_P_1, out => "AMEND".start)
   END_RUNG
   RUNG wire#w1
      { S7_Templates := "SrcType := Int" } GE_Contact(in1 := "BUFF".PROCESS, in2 := 70)
      { S7_Templates := "SrcType := Int" } LE_Contact(in1 := "BUFF".PROCESS, in2 := 80)
      Move(in := "new"."STD ABORT TEMP"[9], out1 => "RETAIN"."SET ABORT TEMP")
      Move(in := "new"."STD OVER TEMP"[9], out1 => "RETAIN"."SET OVERSHOOT")
   END_RUNG
   // the same network as SCL:
   "IEC_Timer_0_DB_81".TON(IN := "AlwaysTRUE" AND ("BUFF".PROCESS = 71) AND ("PV".VACCUM <= "RETAIN"."SET HPHV VCC"),
                           PT := T#1s);
   "IEC_Timer_0_DB_143".TON(IN := "IEC_Timer_0_DB_81".Q, PT := T#1S);
   IF "IEC_Timer_0_DB_143".Q THEN "BUFF".PROCESS := 72; END_IF;
   #_w1 := "IEC_Timer_0_DB_143".Q AND NOT "AlwaysTRUE";
   #_w2 := #_w1 AND NOT "pulse28";   // rising edge
   "pulse28" := #_w1;
   IF #_w2 THEN "AMEND".start := "REVAMP".SEC_P_1; END_IF;
   IF "AlwaysTRUE" AND ("BUFF".PROCESS >= 70) AND ("BUFF".PROCESS <= 80) THEN
       "RETAIN"."SET ABORT TEMP" := "new"."STD ABORT TEMP"[9];
       "RETAIN"."SET OVERSHOOT" := "new"."STD OVER TEMP"[9];
   END_IF;
END_REGION

REGION Network 3
   RUNG wire#powerrail
      Contact( "AlwaysTRUE" )
      { S7_Templates := "SrcType := Int" } EQ_Contact(in1 := "BUFF".PROCESS, in2 := 72)
      wire#w1
      { S7_Templates := "time_type := Time" } "IEC_Timer_0_DB_10".TON(pt := T#1M, et =>)
   END_RUNG
   RUNG wire#w1
      Move(in := "RETAIN"."SET HPHV UP PRESS", out1 => "AUXILIARY"."CHAMBER PRESS")
      Move(in := 121.0, out1 => "AUXILIARY"."CHAMBER TEMP")
   END_RUNG
   RUNG wire#w1
      Contact( "IEC_Timer_0_DB_10".Q )
      wire#w2
      { S7_Templates := "value_type := Int" } "HPHV VCC HOLD".CTU(r := "RESET HPHV VCC", pv := "RETAIN"."SET HPHV VCC HOLD", cv =>)
   END_RUNG
   RUNG wire#w2
      RT_Coil( "IEC_Timer_0_DB_10" )
   END_RUNG
   RUNG wire#w1
      { S7_Templates := "SrcType := Int" } GE_Contact(in1 := "HPHV VCC HOLD".CV, in2 := "RETAIN"."SET HPHV VCC HOLD")
      Move(in := 73, out1 => "BUFF".PROCESS)
   END_RUNG
   RUNG wire#w1
      { S7_Templates := "time_type := Time" } "IEC_Timer_0_DB_85".TON(pt := T#200MS, et =>)
   END_RUNG
   RUNG wire#powerrail
      { S7_Templates := "SrcType := Int" } GE_Contact(in1 := "BUFF".PROCESS, in2 := 74)
      wire#w3
      Coil( "RESET HPHV VCC" )
   END_RUNG
   RUNG wire#powerrail
      { S7_Templates := "SrcType := Int" } EQ_Contact(in1 := "BUFF".PROCESS, in2 := 0)
   END_RUNG wire#w3
   // the same network as SCL:
   #_w1 := "AlwaysTRUE" AND ("BUFF".PROCESS = 72);
   "IEC_Timer_0_DB_10".TON(IN := #_w1, PT := T#1M);
   IF #_w1 THEN
       "AUXILIARY"."CHAMBER PRESS" := "RETAIN"."SET HPHV UP PRESS";
       "AUXILIARY"."CHAMBER TEMP" := 121.0;
   END_IF;
   #_w2 := #_w1 AND "IEC_Timer_0_DB_10".Q;
   "HPHV VCC HOLD".CTU(CU := #_w2, R := "RESET HPHV VCC", PV := "RETAIN"."SET HPHV VCC HOLD");
   IF #_w2 THEN RESET_TIMER("IEC_Timer_0_DB_10"); END_IF;
   IF #_w1 AND ("HPHV VCC HOLD".CV >= "RETAIN"."SET HPHV VCC HOLD") THEN "BUFF".PROCESS := 73; END_IF;
   "IEC_Timer_0_DB_85".TON(IN := #_w1, PT := T#200MS);
   "RESET HPHV VCC" := ("BUFF".PROCESS >= 74) OR ("BUFF".PROCESS = 0);
END_REGION

REGION Network 4
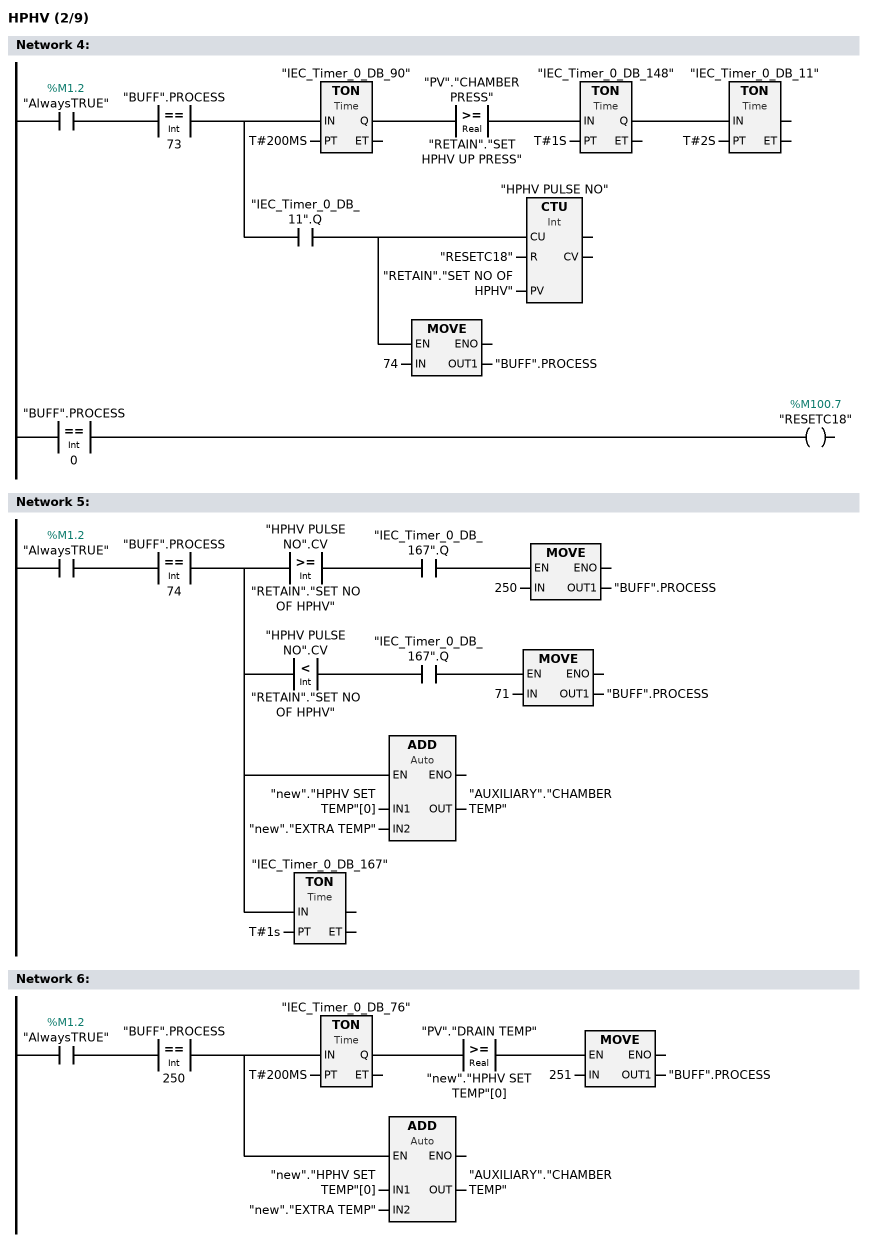
   RUNG wire#powerrail
      Contact( "AlwaysTRUE" )
      { S7_Templates := "SrcType := Int" } EQ_Contact(in1 := "BUFF".PROCESS, in2 := 73)
      wire#w1
      { S7_Templates := "time_type := Time" } "IEC_Timer_0_DB_90".TON(pt := T#200MS, et =>)
      { S7_Templates := "SrcType := Real" } GE_Contact(in1 := "PV"."CHAMBER PRESS", in2 := "RETAIN"."SET HPHV UP PRESS")
      { S7_Templates := "time_type := Time" } "IEC_Timer_0_DB_148".TON(pt := T#1S, et =>)
      { S7_Templates := "time_type := Time" } "IEC_Timer_0_DB_11".TON(pt := T#2S, et =>)
   END_RUNG
   RUNG wire#w1
      Contact( "IEC_Timer_0_DB_11".Q )
      wire#w2
      { S7_Templates := "value_type := Int" } "HPHV PULSE NO".CTU(r := "RESETC18", pv := "RETAIN"."SET NO OF HPHV", cv =>)
   END_RUNG
   RUNG wire#w2
      Move(in := 74, out1 => "BUFF".PROCESS)
   END_RUNG
   RUNG wire#powerrail
      { S7_Templates := "SrcType := Int" } EQ_Contact(in1 := "BUFF".PROCESS, in2 := 0)
      Coil( "RESETC18" )
   END_RUNG
   // the same network as SCL:
   #_w1 := "AlwaysTRUE" AND ("BUFF".PROCESS = 73);
   "IEC_Timer_0_DB_90".TON(IN := #_w1, PT := T#200MS);
   "IEC_Timer_0_DB_148".TON(IN := "IEC_Timer_0_DB_90".Q AND ("PV"."CHAMBER PRESS" >= "RETAIN"."SET HPHV UP PRESS"),
                           PT := T#1S);
   "IEC_Timer_0_DB_11".TON(IN := "IEC_Timer_0_DB_148".Q, PT := T#2S);
   #_w2 := #_w1 AND "IEC_Timer_0_DB_11".Q;
   "HPHV PULSE NO".CTU(CU := #_w2, R := "RESETC18", PV := "RETAIN"."SET NO OF HPHV");
   IF #_w2 THEN "BUFF".PROCESS := 74; END_IF;
   "RESETC18" := "BUFF".PROCESS = 0;
END_REGION

REGION Network 5
   RUNG wire#powerrail
      Contact( "AlwaysTRUE" )
      { S7_Templates := "SrcType := Int" } EQ_Contact(in1 := "BUFF".PROCESS, in2 := 74)
      wire#w1
      { S7_Templates := "SrcType := Int" } GE_Contact(in1 := "HPHV PULSE NO".CV, in2 := "RETAIN"."SET NO OF HPHV")
      Contact( "IEC_Timer_0_DB_167".Q )
      Move(in := 250, out1 => "BUFF".PROCESS)
   END_RUNG
   RUNG wire#w1
      { S7_Templates := "SrcType := Int" } LT_Contact(in1 := "HPHV PULSE NO".CV, in2 := "RETAIN"."SET NO OF HPHV")
      Contact( "IEC_Timer_0_DB_167".Q )
      Move(in := 71, out1 => "BUFF".PROCESS)
   END_RUNG
   RUNG wire#w1
      Add(in1 := "new"."HPHV SET TEMP"[0], in2 := "new"."EXTRA TEMP", out => "AUXILIARY"."CHAMBER TEMP")
   END_RUNG
   RUNG wire#w1
      { S7_Templates := "time_type := Time" } "IEC_Timer_0_DB_167".TON(pt := T#1s, et =>)
   END_RUNG
   // the same network as SCL:
   #_w1 := "AlwaysTRUE" AND ("BUFF".PROCESS = 74);
   IF #_w1 AND ("HPHV PULSE NO".CV >= "RETAIN"."SET NO OF HPHV") AND "IEC_Timer_0_DB_167".Q THEN
       "BUFF".PROCESS := 250;
   END_IF;
   IF #_w1 AND ("HPHV PULSE NO".CV < "RETAIN"."SET NO OF HPHV") AND "IEC_Timer_0_DB_167".Q THEN
       "BUFF".PROCESS := 71;
   END_IF;
   IF #_w1 THEN "AUXILIARY"."CHAMBER TEMP" := "new"."HPHV SET TEMP"[0] + "new"."EXTRA TEMP"; END_IF;
   "IEC_Timer_0_DB_167".TON(IN := #_w1, PT := T#1s);
END_REGION

REGION Network 6
   RUNG wire#powerrail
      Contact( "AlwaysTRUE" )
      { S7_Templates := "SrcType := Int" } EQ_Contact(in1 := "BUFF".PROCESS, in2 := 250)
      wire#w1
      { S7_Templates := "time_type := Time" } "IEC_Timer_0_DB_76".TON(pt := T#200MS, et =>)
      { S7_Templates := "SrcType := Real" } GE_Contact(in1 := "PV"."DRAIN TEMP", in2 := "new"."HPHV SET TEMP"[0])
      Move(in := 251, out1 => "BUFF".PROCESS)
   END_RUNG
   RUNG wire#w1
      Add(in1 := "new"."HPHV SET TEMP"[0], in2 := "new"."EXTRA TEMP", out => "AUXILIARY"."CHAMBER TEMP")
   END_RUNG
   // the same network as SCL:
   #_w1 := "AlwaysTRUE" AND ("BUFF".PROCESS = 250);
   "IEC_Timer_0_DB_76".TON(IN := #_w1, PT := T#200MS);
   IF "IEC_Timer_0_DB_76".Q AND ("PV"."DRAIN TEMP" >= "new"."HPHV SET TEMP"[0]) THEN
       "BUFF".PROCESS := 251;
   END_IF;
   IF #_w1 THEN "AUXILIARY"."CHAMBER TEMP" := "new"."HPHV SET TEMP"[0] + "new"."EXTRA TEMP"; END_IF;
END_REGION

REGION Network 7
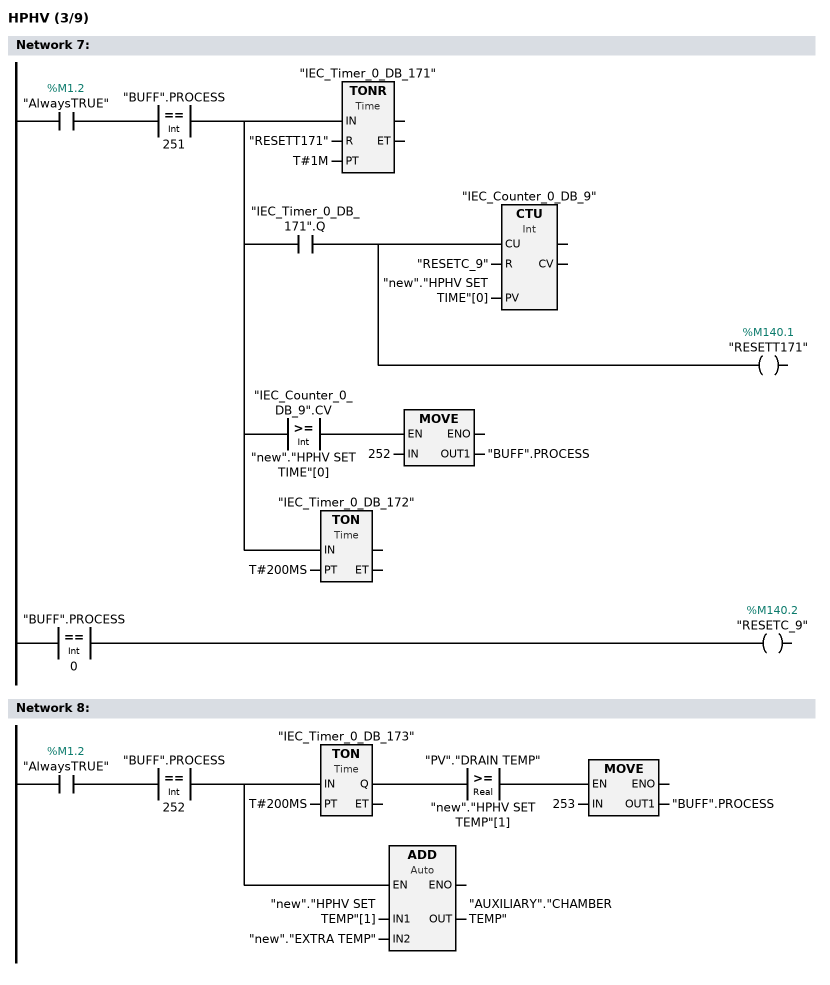
   RUNG wire#powerrail
      Contact( "AlwaysTRUE" )
      { S7_Templates := "SrcType := Int" } EQ_Contact(in1 := "BUFF".PROCESS, in2 := 251)
      wire#w1
      { S7_Templates := "time_type := Time" } "IEC_Timer_0_DB_171".TONR(r := "RESETT171", pt := T#1M, et =>)
   END_RUNG
   RUNG wire#w1
      Contact( "IEC_Timer_0_DB_171".Q )
      wire#w2
      { S7_Templates := "value_type := Int" } "IEC_Counter_0_DB_9".CTU(r := "RESETC_9", pv := "new"."HPHV SET TIME"[0], cv =>)
   END_RUNG
   RUNG wire#w2
      Coil( "RESETT171" )
   END_RUNG
   RUNG wire#w1
      { S7_Templates := "SrcType := Int" } GE_Contact(in1 := "IEC_Counter_0_DB_9".CV, in2 := "new"."HPHV SET TIME"[0])
      Move(in := 252, out1 => "BUFF".PROCESS)
   END_RUNG
   RUNG wire#w1
      { S7_Templates := "time_type := Time" } "IEC_Timer_0_DB_172".TON(pt := T#200MS, et =>)
   END_RUNG
   RUNG wire#powerrail
      { S7_Templates := "SrcType := Int" } EQ_Contact(in1 := "BUFF".PROCESS, in2 := 0)
      Coil( "RESETC_9" )
   END_RUNG
   // the same network as SCL:
   #_w1 := "AlwaysTRUE" AND ("BUFF".PROCESS = 251);
   "IEC_Timer_0_DB_171".TONR(IN := #_w1, R := "RESETT171", PT := T#1M);
   #_w2 := #_w1 AND "IEC_Timer_0_DB_171".Q;
   "IEC_Counter_0_DB_9".CTU(CU := #_w2, R := "RESETC_9", PV := "new"."HPHV SET TIME"[0]);
   "RESETT171" := #_w2;
   IF #_w1 AND ("IEC_Counter_0_DB_9".CV >= "new"."HPHV SET TIME"[0]) THEN "BUFF".PROCESS := 252; END_IF;
   "IEC_Timer_0_DB_172".TON(IN := #_w1, PT := T#200MS);
   "RESETC_9" := "BUFF".PROCESS = 0;
END_REGION

REGION Network 8
   RUNG wire#powerrail
      Contact( "AlwaysTRUE" )
      { S7_Templates := "SrcType := Int" } EQ_Contact(in1 := "BUFF".PROCESS, in2 := 252)
      wire#w1
      { S7_Templates := "time_type := Time" } "IEC_Timer_0_DB_173".TON(pt := T#200MS, et =>)
      { S7_Templates := "SrcType := Real" } GE_Contact(in1 := "PV"."DRAIN TEMP", in2 := "new"."HPHV SET TEMP"[1])
      Move(in := 253, out1 => "BUFF".PROCESS)
   END_RUNG
   RUNG wire#w1
      Add(in1 := "new"."HPHV SET TEMP"[1], in2 := "new"."EXTRA TEMP", out => "AUXILIARY"."CHAMBER TEMP")
   END_RUNG
   // the same network as SCL:
   #_w1 := "AlwaysTRUE" AND ("BUFF".PROCESS = 252);
   "IEC_Timer_0_DB_173".TON(IN := #_w1, PT := T#200MS);
   IF "IEC_Timer_0_DB_173".Q AND ("PV"."DRAIN TEMP" >= "new"."HPHV SET TEMP"[1]) THEN
       "BUFF".PROCESS := 253;
   END_IF;
   IF #_w1 THEN "AUXILIARY"."CHAMBER TEMP" := "new"."HPHV SET TEMP"[1] + "new"."EXTRA TEMP"; END_IF;
END_REGION

REGION Network 9
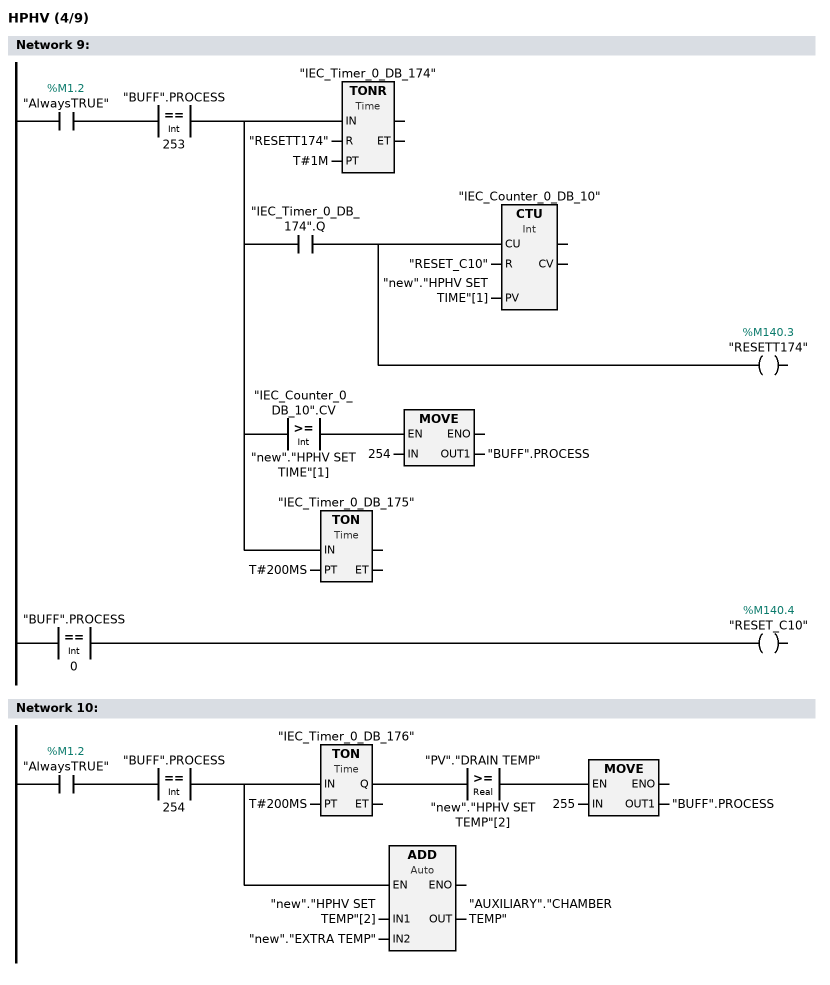
   RUNG wire#powerrail
      Contact( "AlwaysTRUE" )
      { S7_Templates := "SrcType := Int" } EQ_Contact(in1 := "BUFF".PROCESS, in2 := 253)
      wire#w1
      { S7_Templates := "time_type := Time" } "IEC_Timer_0_DB_174".TONR(r := "RESETT174", pt := T#1M, et =>)
   END_RUNG
   RUNG wire#w1
      Contact( "IEC_Timer_0_DB_174".Q )
      wire#w2
      { S7_Templates := "value_type := Int" } "IEC_Counter_0_DB_10".CTU(r := "RESET_C10", pv := "new"."HPHV SET TIME"[1], cv =>)
   END_RUNG
   RUNG wire#w2
      Coil( "RESETT174" )
   END_RUNG
   RUNG wire#w1
      { S7_Templates := "SrcType := Int" } GE_Contact(in1 := "IEC_Counter_0_DB_10".CV, in2 := "new"."HPHV SET TIME"[1])
      Move(in := 254, out1 => "BUFF".PROCESS)
   END_RUNG
   RUNG wire#w1
      { S7_Templates := "time_type := Time" } "IEC_Timer_0_DB_175".TON(pt := T#200MS, et =>)
   END_RUNG
   RUNG wire#powerrail
      { S7_Templates := "SrcType := Int" } EQ_Contact(in1 := "BUFF".PROCESS, in2 := 0)
      Coil( "RESET_C10" )
   END_RUNG
   // the same network as SCL:
   #_w1 := "AlwaysTRUE" AND ("BUFF".PROCESS = 253);
   "IEC_Timer_0_DB_174".TONR(IN := #_w1, R := "RESETT174", PT := T#1M);
   #_w2 := #_w1 AND "IEC_Timer_0_DB_174".Q;
   "IEC_Counter_0_DB_10".CTU(CU := #_w2, R := "RESET_C10", PV := "new"."HPHV SET TIME"[1]);
   "RESETT174" := #_w2;
   IF #_w1 AND ("IEC_Counter_0_DB_10".CV >= "new"."HPHV SET TIME"[1]) THEN "BUFF".PROCESS := 254; END_IF;
   "IEC_Timer_0_DB_175".TON(IN := #_w1, PT := T#200MS);
   "RESET_C10" := "BUFF".PROCESS = 0;
END_REGION

REGION Network 10
   RUNG wire#powerrail
      Contact( "AlwaysTRUE" )
      { S7_Templates := "SrcType := Int" } EQ_Contact(in1 := "BUFF".PROCESS, in2 := 254)
      wire#w1
      { S7_Templates := "time_type := Time" } "IEC_Timer_0_DB_176".TON(pt := T#200MS, et =>)
      { S7_Templates := "SrcType := Real" } GE_Contact(in1 := "PV"."DRAIN TEMP", in2 := "new"."HPHV SET TEMP"[2])
      Move(in := 255, out1 => "BUFF".PROCESS)
   END_RUNG
   RUNG wire#w1
      Add(in1 := "new"."HPHV SET TEMP"[2], in2 := "new"."EXTRA TEMP", out => "AUXILIARY"."CHAMBER TEMP")
   END_RUNG
   // the same network as SCL:
   #_w1 := "AlwaysTRUE" AND ("BUFF".PROCESS = 254);
   "IEC_Timer_0_DB_176".TON(IN := #_w1, PT := T#200MS);
   IF "IEC_Timer_0_DB_176".Q AND ("PV"."DRAIN TEMP" >= "new"."HPHV SET TEMP"[2]) THEN
       "BUFF".PROCESS := 255;
   END_IF;
   IF #_w1 THEN "AUXILIARY"."CHAMBER TEMP" := "new"."HPHV SET TEMP"[2] + "new"."EXTRA TEMP"; END_IF;
END_REGION

REGION Network 11
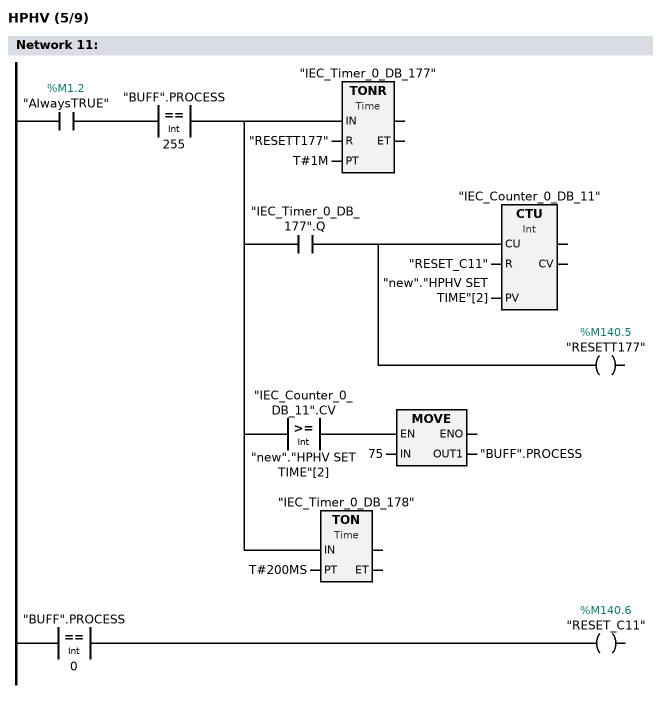
   RUNG wire#powerrail
      Contact( "AlwaysTRUE" )
      { S7_Templates := "SrcType := Int" } EQ_Contact(in1 := "BUFF".PROCESS, in2 := 255)
      wire#w1
      { S7_Templates := "time_type := Time" } "IEC_Timer_0_DB_177".TONR(r := "RESETT177", pt := T#1M, et =>)
   END_RUNG
   RUNG wire#w1
      Contact( "IEC_Timer_0_DB_177".Q )
      wire#w2
      { S7_Templates := "value_type := Int" } "IEC_Counter_0_DB_11".CTU(r := "RESET_C11", pv := "new"."HPHV SET TIME"[2], cv =>)
   END_RUNG
   RUNG wire#w2
      Coil( "RESETT177" )
   END_RUNG
   RUNG wire#w1
      { S7_Templates := "SrcType := Int" } GE_Contact(in1 := "IEC_Counter_0_DB_11".CV, in2 := "new"."HPHV SET TIME"[2])
      Move(in := 75, out1 => "BUFF".PROCESS)
   END_RUNG
   RUNG wire#w1
      { S7_Templates := "time_type := Time" } "IEC_Timer_0_DB_178".TON(pt := T#200MS, et =>)
   END_RUNG
   RUNG wire#powerrail
      { S7_Templates := "SrcType := Int" } EQ_Contact(in1 := "BUFF".PROCESS, in2 := 0)
      Coil( "RESET_C11" )
   END_RUNG
   // the same network as SCL:
   #_w1 := "AlwaysTRUE" AND ("BUFF".PROCESS = 255);
   "IEC_Timer_0_DB_177".TONR(IN := #_w1, R := "RESETT177", PT := T#1M);
   #_w2 := #_w1 AND "IEC_Timer_0_DB_177".Q;
   "IEC_Counter_0_DB_11".CTU(CU := #_w2, R := "RESET_C11", PV := "new"."HPHV SET TIME"[2]);
   "RESETT177" := #_w2;
   IF #_w1 AND ("IEC_Counter_0_DB_11".CV >= "new"."HPHV SET TIME"[2]) THEN "BUFF".PROCESS := 75; END_IF;
   "IEC_Timer_0_DB_178".TON(IN := #_w1, PT := T#200MS);
   "RESET_C11" := "BUFF".PROCESS = 0;
END_REGION

REGION Network 12
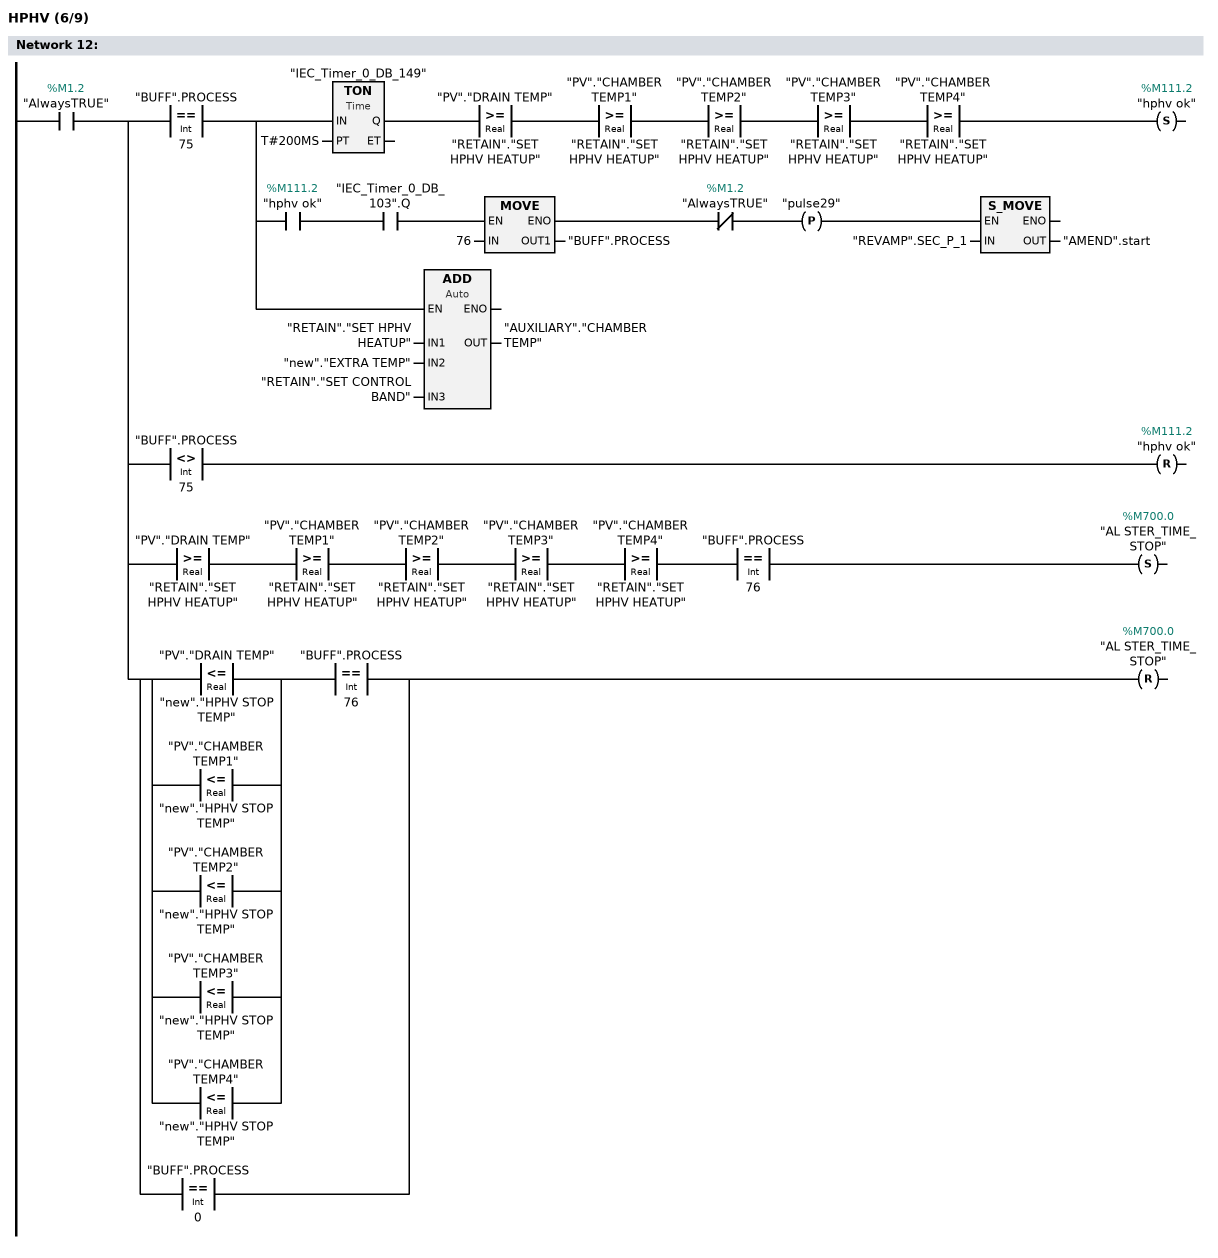
   RUNG wire#powerrail
      Contact( "AlwaysTRUE" )
      wire#w1
      { S7_Templates := "SrcType := Int" } EQ_Contact(in1 := "BUFF".PROCESS, in2 := 75)
      wire#w2
      { S7_Templates := "time_type := Time" } "IEC_Timer_0_DB_149".TON(pt := T#200MS, et =>)
      { S7_Templates := "SrcType := Real" } GE_Contact(in1 := "PV"."DRAIN TEMP", in2 := "RETAIN"."SET HPHV HEATUP")
      { S7_Templates := "SrcType := Real" } GE_Contact(in1 := "PV"."CHAMBER TEMP1", in2 := "RETAIN"."SET HPHV HEATUP")
      { S7_Templates := "SrcType := Real" } GE_Contact(in1 := "PV"."CHAMBER TEMP2", in2 := "RETAIN"."SET HPHV HEATUP")
      { S7_Templates := "SrcType := Real" } GE_Contact(in1 := "PV"."CHAMBER TEMP3", in2 := "RETAIN"."SET HPHV HEATUP")
      { S7_Templates := "SrcType := Real" } GE_Contact(in1 := "PV"."CHAMBER TEMP4", in2 := "RETAIN"."SET HPHV HEATUP")
      S_Coil( "hphv ok" )
   END_RUNG
   RUNG wire#w2
      Contact( "hphv ok" )
      Contact( "IEC_Timer_0_DB_103".Q )
      Move(in := 76, out1 => "BUFF".PROCESS)
      I_Contact( "AlwaysTRUE" )
      P_Trig( "pulse29" )
      S_Move(in := "REVAMP".SEC_P_1, out => "AMEND".start)
   END_RUNG
   RUNG wire#w2
      Add(in1 := "RETAIN"."SET HPHV HEATUP", in2 := "new"."EXTRA TEMP", in3 := "RETAIN"."SET CONTROL BAND", out => "AUXILIARY"."CHAMBER TEMP")
   END_RUNG
   RUNG wire#w1
      { S7_Templates := "SrcType := Int" } NE_Contact(in1 := "BUFF".PROCESS, in2 := 75)
      R_Coil( "hphv ok" )
   END_RUNG
   RUNG wire#w1
      { S7_Templates := "SrcType := Real" } GE_Contact(in1 := "PV"."DRAIN TEMP", in2 := "RETAIN"."SET HPHV HEATUP")
      { S7_Templates := "SrcType := Real" } GE_Contact(in1 := "PV"."CHAMBER TEMP1", in2 := "RETAIN"."SET HPHV HEATUP")
      { S7_Templates := "SrcType := Real" } GE_Contact(in1 := "PV"."CHAMBER TEMP2", in2 := "RETAIN"."SET HPHV HEATUP")
      { S7_Templates := "SrcType := Real" } GE_Contact(in1 := "PV"."CHAMBER TEMP3", in2 := "RETAIN"."SET HPHV HEATUP")
      { S7_Templates := "SrcType := Real" } GE_Contact(in1 := "PV"."CHAMBER TEMP4", in2 := "RETAIN"."SET HPHV HEATUP")
      { S7_Templates := "SrcType := Int" } EQ_Contact(in1 := "BUFF".PROCESS, in2 := 76)
      S_Coil( "AL STER_TIME_STOP" )
   END_RUNG
   RUNG wire#w1
      { S7_Templates := "SrcType := Real" } LE_Contact(in1 := "PV"."DRAIN TEMP", in2 := "new"."HPHV STOP TEMP")
      wire#w3
      { S7_Templates := "SrcType := Int" } EQ_Contact(in1 := "BUFF".PROCESS, in2 := 76)
      wire#w4
      R_Coil( "AL STER_TIME_STOP" )
   END_RUNG
   RUNG wire#w1
      { S7_Templates := "SrcType := Real" } LE_Contact(in1 := "PV"."CHAMBER TEMP1", in2 := "new"."HPHV STOP TEMP")
   END_RUNG wire#w3
   RUNG wire#w1
      { S7_Templates := "SrcType := Real" } LE_Contact(in1 := "PV"."CHAMBER TEMP2", in2 := "new"."HPHV STOP TEMP")
   END_RUNG wire#w3
   RUNG wire#w1
      { S7_Templates := "SrcType := Real" } LE_Contact(in1 := "PV"."CHAMBER TEMP3", in2 := "new"."HPHV STOP TEMP")
   END_RUNG wire#w3
   RUNG wire#w1
      { S7_Templates := "SrcType := Real" } LE_Contact(in1 := "PV"."CHAMBER TEMP4", in2 := "new"."HPHV STOP TEMP")
   END_RUNG wire#w3
   RUNG wire#w1
      { S7_Templates := "SrcType := Int" } EQ_Contact(in1 := "BUFF".PROCESS, in2 := 0)
   END_RUNG wire#w4
   // the same network as SCL:
   #_w1 := "AlwaysTRUE" AND ("BUFF".PROCESS = 75);
   "IEC_Timer_0_DB_149".TON(IN := #_w1, PT := T#200MS);
   IF "IEC_Timer_0_DB_149".Q AND ("PV"."DRAIN TEMP" >= "RETAIN"."SET HPHV HEATUP") AND ("PV"."CHAMBER TEMP1" >= "RETAIN"."SET HPHV HEATUP") AND ("PV"."CHAMBER TEMP2" >= "RETAIN"."SET HPHV HEATUP") AND ("PV"."CHAMBER TEMP3" >= "RETAIN"."SET HPHV HEATUP") AND ("PV"."CHAMBER TEMP4" >= "RETAIN"."SET HPHV HEATUP") THEN
       "hphv ok" := TRUE;
   END_IF;
   #_w2 := #_w1 AND "hphv ok" AND "IEC_Timer_0_DB_103".Q;
   IF #_w2 THEN "BUFF".PROCESS := 76; END_IF;
   #_w3 := #_w2 AND NOT "AlwaysTRUE";
   #_w4 := #_w3 AND NOT "pulse29";   // rising edge
   "pulse29" := #_w3;
   IF #_w4 THEN "AMEND".start := "REVAMP".SEC_P_1; END_IF;
   IF #_w1 THEN
       "AUXILIARY"."CHAMBER TEMP" := "RETAIN"."SET HPHV HEATUP" + "new"."EXTRA TEMP" + "RETAIN"."SET CONTROL BAND";
   END_IF;
   IF "AlwaysTRUE" AND ("BUFF".PROCESS <> 75) THEN "hphv ok" := FALSE; END_IF;
   IF "AlwaysTRUE" AND ("PV"."DRAIN TEMP" >= "RETAIN"."SET HPHV HEATUP") AND ("PV"."CHAMBER TEMP1" >= "RETAIN"."SET HPHV HEATUP") AND ("PV"."CHAMBER TEMP2" >= "RETAIN"."SET HPHV HEATUP") AND ("PV"."CHAMBER TEMP3" >= "RETAIN"."SET HPHV HEATUP") AND ("PV"."CHAMBER TEMP4" >= "RETAIN"."SET HPHV HEATUP") AND ("BUFF".PROCESS = 76) THEN
       "AL STER_TIME_STOP" := TRUE;
   END_IF;
   IF "AlwaysTRUE" AND (((("PV"."DRAIN TEMP" <= "new"."HPHV STOP TEMP") OR ("PV"."CHAMBER TEMP1" <= "new"."HPHV STOP TEMP") OR ("PV"."CHAMBER TEMP2" <= "new"."HPHV STOP TEMP") OR ("PV"."CHAMBER TEMP3" <= "new"."HPHV STOP TEMP") OR ("PV"."CHAMBER TEMP4" <= "new"."HPHV STOP TEMP")) AND ("BUFF".PROCESS = 76)) OR ("BUFF".PROCESS = 0)) THEN
       "AL STER_TIME_STOP" := FALSE;
   END_IF;
END_REGION

REGION Network 13
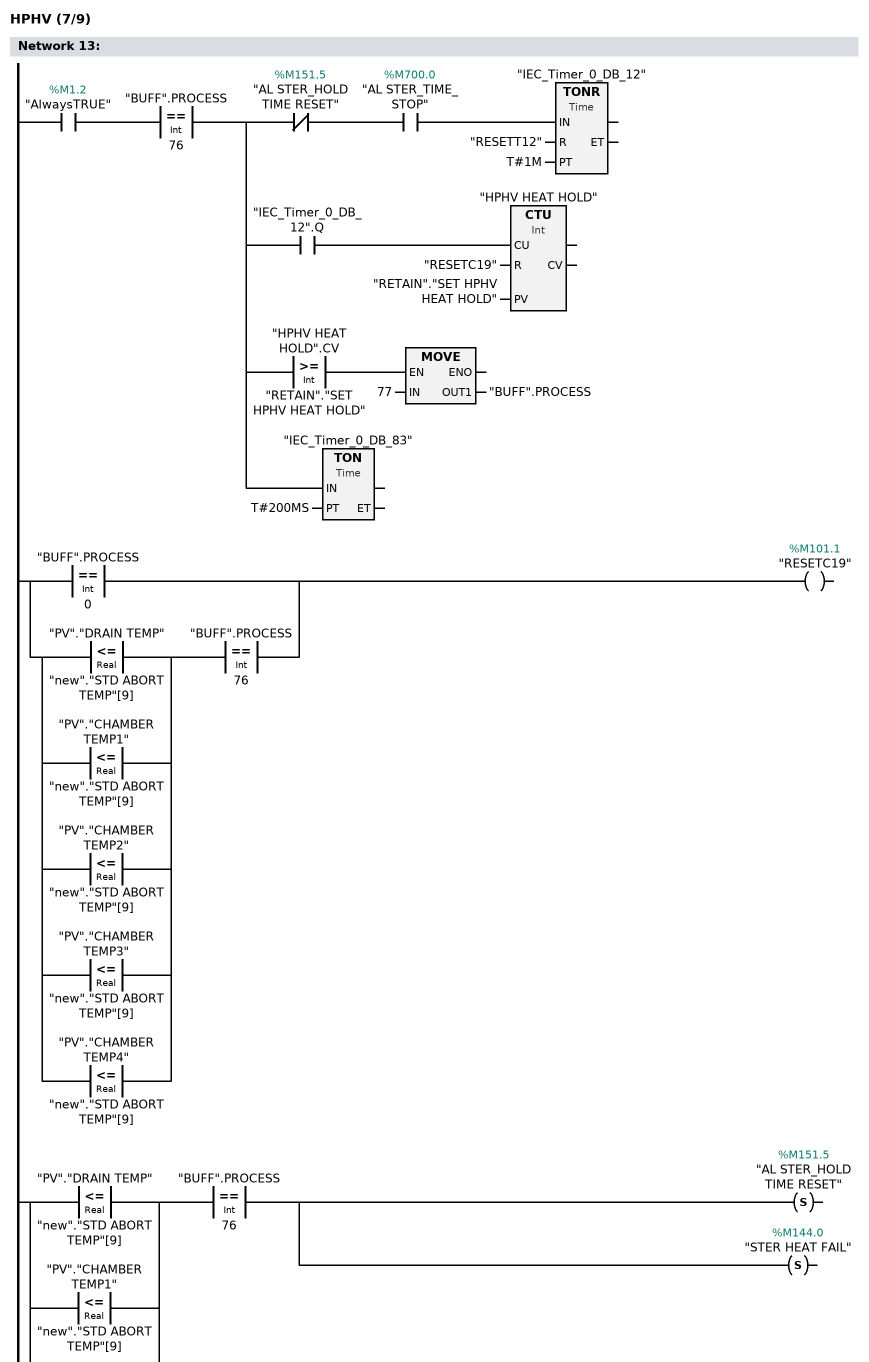
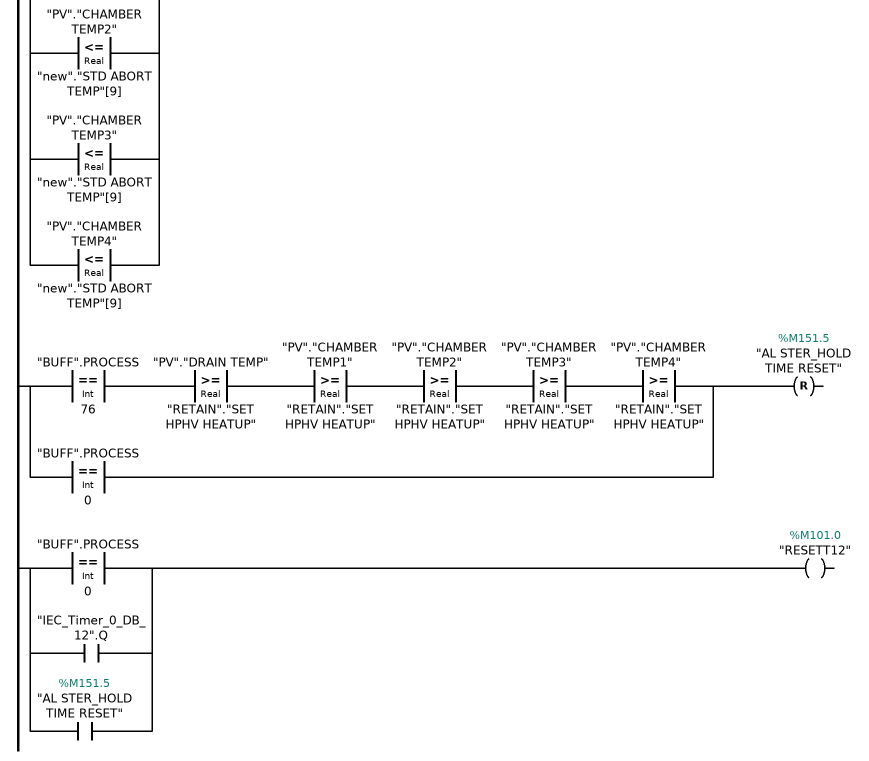
   RUNG wire#powerrail
      Contact( "AlwaysTRUE" )
      { S7_Templates := "SrcType := Int" } EQ_Contact(in1 := "BUFF".PROCESS, in2 := 76)
      wire#w1
      I_Contact( "AL STER_HOLD TIME RESET" )
      Contact( "AL STER_TIME_STOP" )
      { S7_Templates := "time_type := Time" } "IEC_Timer_0_DB_12".TONR(r := "RESETT12", pt := T#1M, et =>)
   END_RUNG
   RUNG wire#w1
      Contact( "IEC_Timer_0_DB_12".Q )
      { S7_Templates := "value_type := Int" } "HPHV HEAT HOLD".CTU(r := "RESETC19", pv := "RETAIN"."SET HPHV HEAT HOLD", cv =>)
   END_RUNG
   RUNG wire#w1
      { S7_Templates := "SrcType := Int" } GE_Contact(in1 := "HPHV HEAT HOLD".CV, in2 := "RETAIN"."SET HPHV HEAT HOLD")
      Move(in := 77, out1 => "BUFF".PROCESS)
   END_RUNG
   RUNG wire#w1
      { S7_Templates := "time_type := Time" } "IEC_Timer_0_DB_83".TON(pt := T#200MS, et =>)
   END_RUNG
   RUNG wire#powerrail
      { S7_Templates := "SrcType := Int" } EQ_Contact(in1 := "BUFF".PROCESS, in2 := 0)
      wire#w2
      Coil( "RESETC19" )
   END_RUNG
   RUNG wire#powerrail
      { S7_Templates := "SrcType := Real" } LE_Contact(in1 := "PV"."DRAIN TEMP", in2 := "new"."STD ABORT TEMP"[9])
      wire#w3
      { S7_Templates := "SrcType := Int" } EQ_Contact(in1 := "BUFF".PROCESS, in2 := 76)
   END_RUNG wire#w2
   RUNG wire#powerrail
      { S7_Templates := "SrcType := Real" } LE_Contact(in1 := "PV"."CHAMBER TEMP1", in2 := "new"."STD ABORT TEMP"[9])
   END_RUNG wire#w3
   RUNG wire#powerrail
      { S7_Templates := "SrcType := Real" } LE_Contact(in1 := "PV"."CHAMBER TEMP2", in2 := "new"."STD ABORT TEMP"[9])
   END_RUNG wire#w3
   RUNG wire#powerrail
      { S7_Templates := "SrcType := Real" } LE_Contact(in1 := "PV"."CHAMBER TEMP3", in2 := "new"."STD ABORT TEMP"[9])
   END_RUNG wire#w3
   RUNG wire#powerrail
      { S7_Templates := "SrcType := Real" } LE_Contact(in1 := "PV"."CHAMBER TEMP4", in2 := "new"."STD ABORT TEMP"[9])
   END_RUNG wire#w3
   RUNG wire#powerrail
      { S7_Templates := "SrcType := Real" } LE_Contact(in1 := "PV"."DRAIN TEMP", in2 := "new"."STD ABORT TEMP"[9])
      wire#w4
      { S7_Templates := "SrcType := Int" } EQ_Contact(in1 := "BUFF".PROCESS, in2 := 76)
      wire#w5
      S_Coil( "AL STER_HOLD TIME RESET" )
   END_RUNG
   RUNG wire#powerrail
      { S7_Templates := "SrcType := Real" } LE_Contact(in1 := "PV"."CHAMBER TEMP1", in2 := "new"."STD ABORT TEMP"[9])
   END_RUNG wire#w4
   RUNG wire#powerrail
      { S7_Templates := "SrcType := Real" } LE_Contact(in1 := "PV"."CHAMBER TEMP2", in2 := "new"."STD ABORT TEMP"[9])
   END_RUNG wire#w4
   RUNG wire#powerrail
      { S7_Templates := "SrcType := Real" } LE_Contact(in1 := "PV"."CHAMBER TEMP3", in2 := "new"."STD ABORT TEMP"[9])
   END_RUNG wire#w4
   RUNG wire#powerrail
      { S7_Templates := "SrcType := Real" } LE_Contact(in1 := "PV"."CHAMBER TEMP4", in2 := "new"."STD ABORT TEMP"[9])
   END_RUNG wire#w4
   RUNG wire#w5
      S_Coil( "STER HEAT FAIL" )
   END_RUNG
   RUNG wire#powerrail
      { S7_Templates := "SrcType := Int" } EQ_Contact(in1 := "BUFF".PROCESS, in2 := 76)
      { S7_Templates := "SrcType := Real" } GE_Contact(in1 := "PV"."DRAIN TEMP", in2 := "RETAIN"."SET HPHV HEATUP")
      { S7_Templates := "SrcType := Real" } GE_Contact(in1 := "PV"."CHAMBER TEMP1", in2 := "RETAIN"."SET HPHV HEATUP")
      { S7_Templates := "SrcType := Real" } GE_Contact(in1 := "PV"."CHAMBER TEMP2", in2 := "RETAIN"."SET HPHV HEATUP")
      { S7_Templates := "SrcType := Real" } GE_Contact(in1 := "PV"."CHAMBER TEMP3", in2 := "RETAIN"."SET HPHV HEATUP")
      { S7_Templates := "SrcType := Real" } GE_Contact(in1 := "PV"."CHAMBER TEMP4", in2 := "RETAIN"."SET HPHV HEATUP")
      wire#w6
      R_Coil( "AL STER_HOLD TIME RESET" )
   END_RUNG
   RUNG wire#powerrail
      { S7_Templates := "SrcType := Int" } EQ_Contact(in1 := "BUFF".PROCESS, in2 := 0)
   END_RUNG wire#w6
   RUNG wire#powerrail
      { S7_Templates := "SrcType := Int" } EQ_Contact(in1 := "BUFF".PROCESS, in2 := 0)
      wire#w7
      Coil( "RESETT12" )
   END_RUNG
   RUNG wire#powerrail
      Contact( "IEC_Timer_0_DB_12".Q )
   END_RUNG wire#w7
   RUNG wire#powerrail
      Contact( "AL STER_HOLD TIME RESET" )
   END_RUNG wire#w7
   // the same network as SCL:
   #_w1 := "AlwaysTRUE" AND ("BUFF".PROCESS = 76);
   "IEC_Timer_0_DB_12".TONR(IN := #_w1 AND NOT "AL STER_HOLD TIME RESET" AND "AL STER_TIME_STOP",
                           R := "RESETT12",
                           PT := T#1M);
   "HPHV HEAT HOLD".CTU(CU := #_w1 AND "IEC_Timer_0_DB_12".Q,
                        R := "RESETC19",
                        PV := "RETAIN"."SET HPHV HEAT HOLD");
   IF #_w1 AND ("HPHV HEAT HOLD".CV >= "RETAIN"."SET HPHV HEAT HOLD") THEN "BUFF".PROCESS := 77; END_IF;
   "IEC_Timer_0_DB_83".TON(IN := #_w1, PT := T#200MS);
   "RESETC19" := ("BUFF".PROCESS = 0) OR ((("PV"."DRAIN TEMP" <= "new"."STD ABORT TEMP"[9]) OR ("PV"."CHAMBER TEMP1" <= "new"."STD ABORT TEMP"[9]) OR ("PV"."CHAMBER TEMP2" <= "new"."STD ABORT TEMP"[9]) OR ("PV"."CHAMBER TEMP3" <= "new"."STD ABORT TEMP"[9]) OR ("PV"."CHAMBER TEMP4" <= "new"."STD ABORT TEMP"[9])) AND ("BUFF".PROCESS = 76));
   IF (("PV"."DRAIN TEMP" <= "new"."STD ABORT TEMP"[9]) OR ("PV"."CHAMBER TEMP1" <= "new"."STD ABORT TEMP"[9]) OR ("PV"."CHAMBER TEMP2" <= "new"."STD ABORT TEMP"[9]) OR ("PV"."CHAMBER TEMP3" <= "new"."STD ABORT TEMP"[9]) OR ("PV"."CHAMBER TEMP4" <= "new"."STD ABORT TEMP"[9])) AND ("BUFF".PROCESS = 76) THEN
       "AL STER_HOLD TIME RESET" := TRUE;
       "STER HEAT FAIL" := TRUE;
   END_IF;
   IF (("BUFF".PROCESS = 76) AND ("PV"."DRAIN TEMP" >= "RETAIN"."SET HPHV HEATUP") AND ("PV"."CHAMBER TEMP1" >= "RETAIN"."SET HPHV HEATUP") AND ("PV"."CHAMBER TEMP2" >= "RETAIN"."SET HPHV HEATUP") AND ("PV"."CHAMBER TEMP3" >= "RETAIN"."SET HPHV HEATUP") AND ("PV"."CHAMBER TEMP4" >= "RETAIN"."SET HPHV HEATUP")) OR ("BUFF".PROCESS = 0) THEN
       "AL STER_HOLD TIME RESET" := FALSE;
   END_IF;
   "RESETT12" := ("BUFF".PROCESS = 0) OR "IEC_Timer_0_DB_12".Q OR "AL STER_HOLD TIME RESET";
END_REGION

REGION Network 14
